// Mitsubishi GX Works2 project: china press #3 kontroller   PLC: Q04UDEH

// task MAIN (event TRUE, interval 0, priority 31): MAIN
// task MAIN1 (event TRUE, interval 0, priority 31): MAIN1_Block000
// task SFC (event TRUE, interval 0, priority 31): SFC_Block000, SFC_Block001, SFC_Block003, SFC_Block004, SFC_Block005, SFC_Block006

PROGRAM MAIN
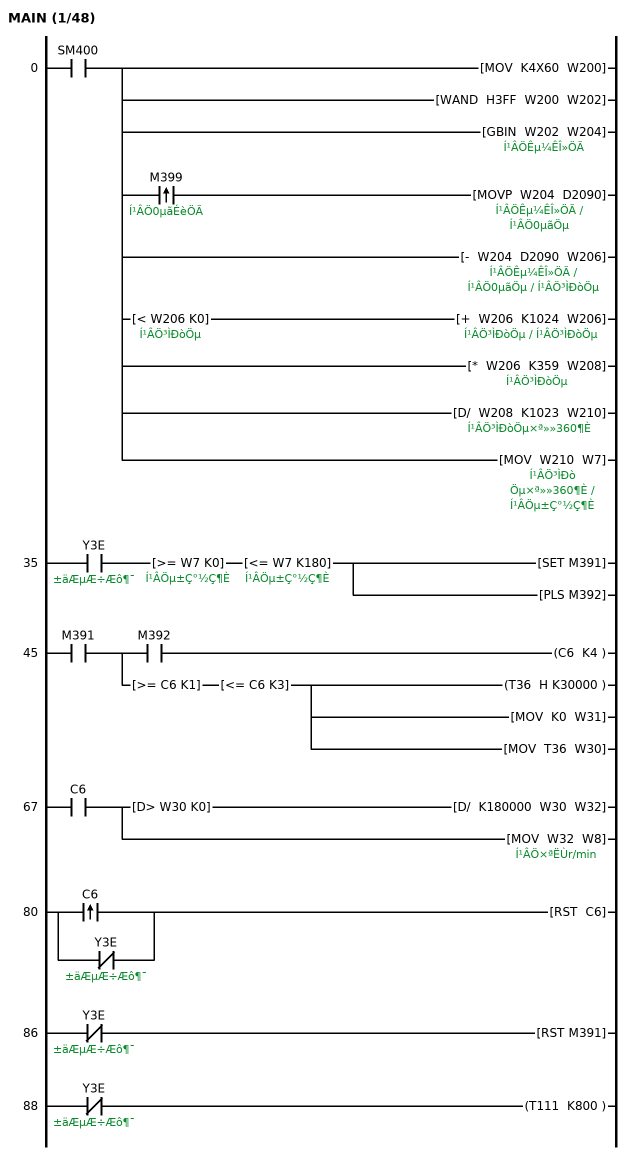
0     LD      SM400
      MOV     K4X60 W200  ; ¾øµØÖµ±àÂëÆ÷1
      WAND    H3FF W200 W202
      GBIN    W202 W204  ; Í¹ÂÖÊµ¼ÊÎ»ÖÃ
      MPS
      ANDP    M399  ; Í¹ÂÖ0µãÉèÖÃ
      MOVP    W204 D2090  ; Í¹ÂÖ0µãÖµ
      MPP
      -       W204 D2090 W206  ; Í¹ÂÖ³ÌÐòÖµ
      MPS
      AND<    W206 K0  ; Í¹ÂÖ³ÌÐòÖµ
      +       W206 K1024 W206
      MPP
      *       W206 K359 W208
      D/      W208 K1023 W210  ; Í¹ÂÖ³ÌÐòÖµ×ª»»360¶È
      MOV     W210 W7  ; Í¹ÂÖµ±Ç°½Ç¶È
35    LD      Y3E  ; ±äÆµÆ÷Æô¶¯
      AND>=   W7 K0  ; Í¹ÂÖµ±Ç°½Ç¶È
      AND<=   W7 K180  ; Í¹ÂÖµ±Ç°½Ç¶È
      SET     M391
      PLS     M392
45    LD      M391
      MPS
      AND     M392
      OUT     C6 K4
      MPP
      AND>=   C6 K1
      AND<=   C6 K3
      OUTH    T36 K30000
      MOV     K0 W31
      MOV     T36 W30
67    LD      C6
      MPS
      ANDD>   W30 K0
      D/      K180000 W30 W32
      MPP
      MOV     W32 W8  ; Í¹ÂÖ×ªËÙr/min
80    LDP     C6
      ORI     Y3E  ; ±äÆµÆ÷Æô¶¯
      RST     C6
86    LDI     Y3E  ; ±äÆµÆ÷Æô¶¯
      RST     M391
88    LDI     Y3E  ; ±äÆµÆ÷Æô¶¯
      OUT     T111 K800
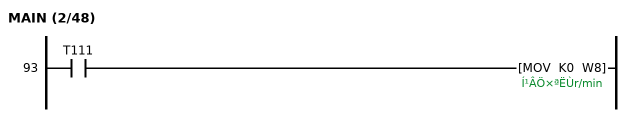
93    LD      T111
      MOV     K0 W8
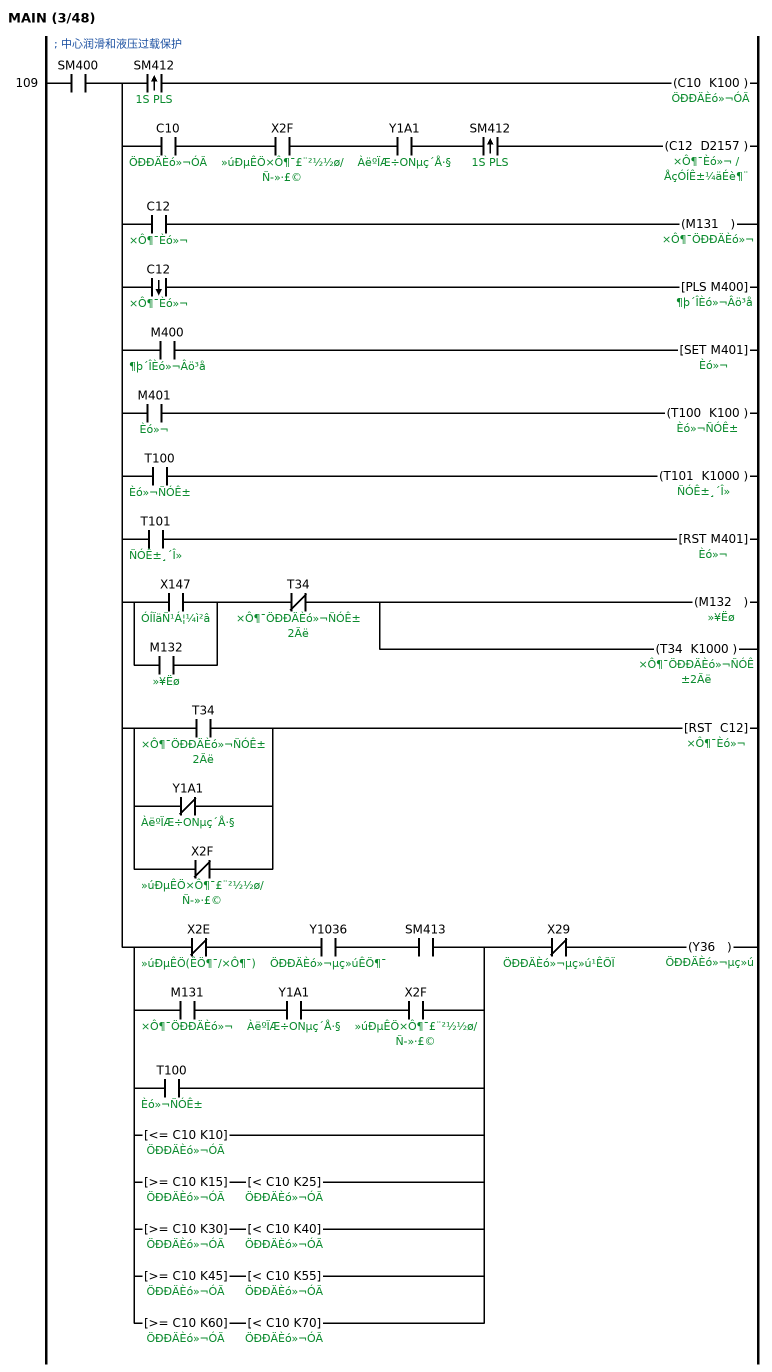
; 中心润滑和液压过载保护
109   LD      SM400
      MPS
      ANDP    SM412  ; 1S PLS
      OUT     C10 K100  ; ÖÐÐÄÈó»¬ÓÃ
      MRD
      AND     C10  ; ÖÐÐÄÈó»¬ÓÃ
      AND     X2F  ; »úÐµÊÖ×Ô¶¯£¨²½½ø/Ñ­»·£©
      AND     Y1A1  ; ÀëºÏÆ÷ONµç´Å·§
      ANDP    SM412  ; 1S PLS
      OUT     C12 D2157  ; ×Ô¶¯Èó»¬ / ÅçÓÍÊ±¼äÉè¶¨
      MRD
      AND     C12  ; ×Ô¶¯Èó»¬
      OUT     M131  ; ×Ô¶¯ÖÐÐÄÈó»¬
      MRD
      ANDF    C12  ; ×Ô¶¯Èó»¬
      PLS     M400  ; ¶þ´ÎÈó»¬Âö³å
      MRD
      AND     M400  ; ¶þ´ÎÈó»¬Âö³å
      SET     M401  ; Èó»¬
      MRD
      AND     M401  ; Èó»¬
      OUT     T100 K100  ; Èó»¬ÑÓÊ±
      MRD
      AND     T100  ; Èó»¬ÑÓÊ±
      OUT     T101 K1000  ; ÑÓÊ±¸´Î»
      MRD
      AND     T101  ; ÑÓÊ±¸´Î»
      RST     M401  ; Èó»¬
      MRD
      LD      X147  ; ÓÍÏäÑ¹Á¦¼ì²â
      OR      M132  ; »¥Ëø
      ANB
      ANI     T34  ; ×Ô¶¯ÖÐÐÄÈó»¬ÑÓÊ±2Ãë
      OUT     M132  ; »¥Ëø
      OUT     T34 K1000  ; ×Ô¶¯ÖÐÐÄÈó»¬ÑÓÊ±2Ãë
      MRD
      LD      T34  ; ×Ô¶¯ÖÐÐÄÈó»¬ÑÓÊ±2Ãë
      ORI     Y1A1  ; ÀëºÏÆ÷ONµç´Å·§
      ORI     X2F  ; »úÐµÊÖ×Ô¶¯£¨²½½ø/Ñ­»·£©
      ANB
      RST     C12  ; ×Ô¶¯Èó»¬
      MPP
      LDI     X2E  ; »úÐµÊÖ(ÊÖ¶¯/×Ô¶¯)
      AND     Y1036  ; ÖÐÐÄÈó»¬µç»úÊÖ¶¯
      AND     SM413
      LD      M131  ; ×Ô¶¯ÖÐÐÄÈó»¬
      AND     Y1A1  ; ÀëºÏÆ÷ONµç´Å·§
      AND     X2F  ; »úÐµÊÖ×Ô¶¯£¨²½½ø/Ñ­»·£©
      ORB
      OR      T100  ; Èó»¬ÑÓÊ±
      OR<=    C10 K10  ; ÖÐÐÄÈó»¬ÓÃ
      LD>=    C10 K15  ; ÖÐÐÄÈó»¬ÓÃ
      AND<    C10 K25  ; ÖÐÐÄÈó»¬ÓÃ
      ORB
      LD>=    C10 K30  ; ÖÐÐÄÈó»¬ÓÃ
      AND<    C10 K40  ; ÖÐÐÄÈó»¬ÓÃ
      ORB
      LD>=    C10 K45  ; ÖÐÐÄÈó»¬ÓÃ
      AND<    C10 K55  ; ÖÐÐÄÈó»¬ÓÃ
      ORB
      LD>=    C10 K60  ; ÖÐÐÄÈó»¬ÓÃ
      AND<    C10 K70  ; ÖÐÐÄÈó»¬ÓÃ
      ORB
      ANB
      ANI     X29  ; ÖÐÐÄÈó»¬µç»ú¹ÊÕÏ
      OUT     Y36  ; ÖÐÐÄÈó»¬µç»ú
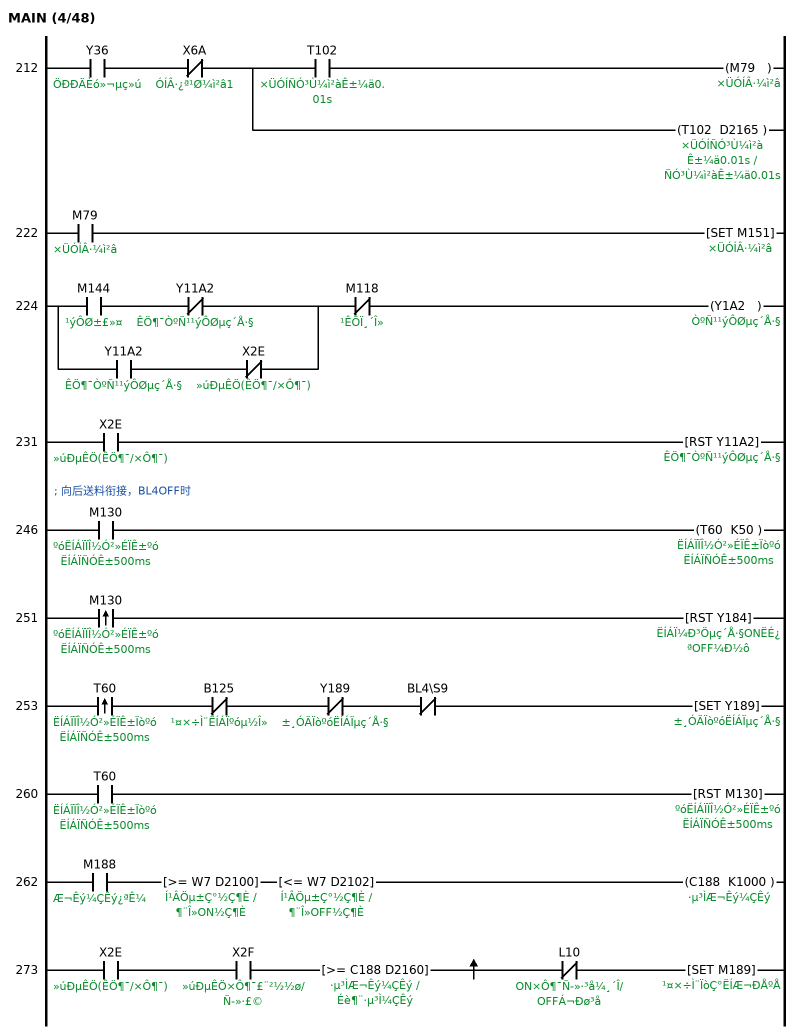
212   LD      Y36  ; ÖÐÐÄÈó»¬µç»ú
      ANI     X6A  ; ÓÍÂ·¿ª¹Ø¼ì²â1
      MPS
      AND     T102  ; ×ÜÓÍÑÓ³Ù¼ì²àÊ±¼ä0.01s
      OUT     M79  ; ×ÜÓÍÂ·¼ì²â
      MPP
      OUT     T102 D2165  ; ×ÜÓÍÑÓ³Ù¼ì²àÊ±¼ä0.01s / ÑÓ³Ù¼ì²àÊ±¼ä0.01s
222   LD      M79  ; ×ÜÓÍÂ·¼ì²â
      SET     M151  ; ×ÜÓÍÂ·¼ì²â
224   LD      M144  ; ¹ýÔØ±£»¤
      ANI     Y11A2  ; ÊÖ¶¯ÒºÑ¹¹ýÔØµç´Å·§
      LD      Y11A2  ; ÊÖ¶¯ÒºÑ¹¹ýÔØµç´Å·§
      ANI     X2E  ; »úÐµÊÖ(ÊÖ¶¯/×Ô¶¯)
      ORB
      ANI     M118  ; ¹ÊÕÏ¸´Î»
      OUT     Y1A2  ; ÒºÑ¹¹ýÔØµç´Å·§
231   LD      X2E  ; »úÐµÊÖ(ÊÖ¶¯/×Ô¶¯)
      RST     Y11A2  ; ÊÖ¶¯ÒºÑ¹¹ýÔØµç´Å·§
; 向后送料衔接，BL4OFF时
246   LD      M130  ; ºóËÍÁÏÏÎ½Ó²»ÉÏÊ±ºóËÍÁÏÑÓÊ±500ms
      OUT     T60 K50  ; ËÍÁÏÏÎ½Ó²»ÉÏÊ±ÏòºóËÍÁÏÑÓÊ±500ms
251   LDP     M130  ; ºóËÍÁÏÏÎ½Ó²»ÉÏÊ±ºóËÍÁÏÑÓÊ±500ms
      RST     Y184  ; ËÍÁÏ¼Ð³Öµç´Å·§ONËÉ¿ªOFF¼Ð½ô
253   LDP     T60  ; ËÍÁÏÏÎ½Ó²»ÉÏÊ±ÏòºóËÍÁÏÑÓÊ±500ms
      ANI     B125  ; ¹¤×÷Ì¨ËÍÁÏºóµ½Î»
      ANI     Y189  ; ±¸ÓÃÏòºóËÍÁÏµç´Å·§
      ANI     BL4\S9
      SET     Y189  ; ±¸ÓÃÏòºóËÍÁÏµç´Å·§
260   LD      T60  ; ËÍÁÏÏÎ½Ó²»ÉÏÊ±ÏòºóËÍÁÏÑÓÊ±500ms
      RST     M130  ; ºóËÍÁÏÏÎ½Ó²»ÉÏÊ±ºóËÍÁÏÑÓÊ±500ms
262   LD      M188  ; Æ¬Êý¼ÇÊý¿ªÊ¼
      AND>=   W7 D2100  ; Í¹ÂÖµ±Ç°½Ç¶È / ¶¨Î»ON½Ç¶È
      AND<=   W7 D2102  ; Í¹ÂÖµ±Ç°½Ç¶È / ¶¨Î»OFF½Ç¶È
      OUT     C188 K1000  ; ·µ³ÌÆ¬Êý¼ÇÊý
273   LD      X2E  ; »úÐµÊÖ(ÊÖ¶¯/×Ô¶¯)
      AND     X2F  ; »úÐµÊÖ×Ô¶¯£¨²½½ø/Ñ­»·£©
      AND>=   C188 D2160  ; ·µ³ÌÆ¬Êý¼ÇÊý / Éè¶¨·µ³Ì¼ÇÊý
      MEP
      ANI     L10  ; ON×Ô¶¯Ñ­»·³å¼¸´Î/OFFÁ¬Ðø³å
      SET     M189  ; ¹¤×÷Ì¨ÏòÇ°ËÍÆ¬ÐÅºÅ
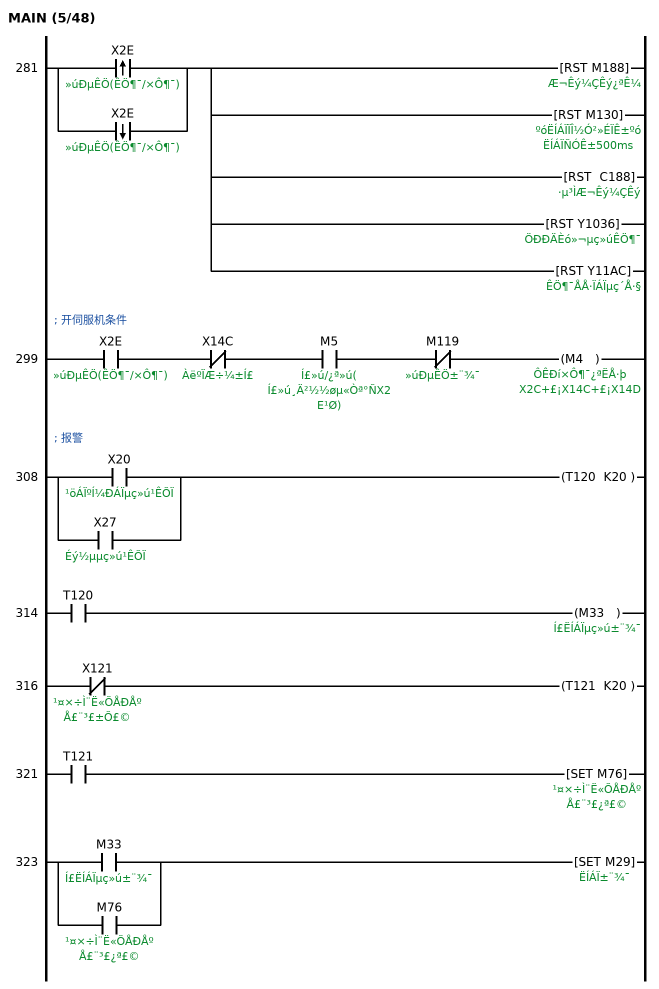
281   LDP     X2E  ; »úÐµÊÖ(ÊÖ¶¯/×Ô¶¯)
      ORF     X2E  ; »úÐµÊÖ(ÊÖ¶¯/×Ô¶¯)
      RST     M188  ; Æ¬Êý¼ÇÊý¿ªÊ¼
      RST     M130  ; ºóËÍÁÏÏÎ½Ó²»ÉÏÊ±ºóËÍÁÏÑÓÊ±500ms
      RST     C188  ; ·µ³ÌÆ¬Êý¼ÇÊý
      RST     Y1036  ; ÖÐÐÄÈó»¬µç»úÊÖ¶¯
      RST     Y11AC  ; ÊÖ¶¯ÅÅ·ÏÁÏµç´Å·§
; 开伺服机条件
299   LD      X2E  ; »úÐµÊÖ(ÊÖ¶¯/×Ô¶¯)
      ANI     X14C  ; ÀëºÏÆ÷¼±Í£
      AND     M5  ; Í£»ú/¿ª»ú(Í£»ú¸Ä²½½øµ«Òª°ÑX2E¹Ø)
      ANI     M119  ; »úÐµÊÖ±¨¾¯
      OUT     M4  ; ÔÊÐí×Ô¶¯¿ªËÅ·þX2C+£¡X14C+£¡X14D
; 报警
308   LD      X20  ; ¹öÁÏºÍ¼ÐÁÏµç»ú¹ÊÕÏ
      OR      X27  ; Éý½µµç»ú¹ÊÕÏ
      OUT     T120 K20
314   LD      T120
      OUT     M33  ; Í£ËÍÁÏµç»ú±¨¾¯
316   LDI     X121  ; ¹¤×÷Ì¨Ë«ÕÅÐÅºÅ£¨³£±Õ£©
      OUT     T121 K20
321   LD      T121
      SET     M76  ; ¹¤×÷Ì¨Ë«ÕÅÐÅºÅ£¨³£¿ª£©
323   LD      M33  ; Í£ËÍÁÏµç»ú±¨¾¯
      OR      M76  ; ¹¤×÷Ì¨Ë«ÕÅÐÅºÅ£¨³£¿ª£©
      SET     M29  ; ËÍÁÏ±¨¾¯
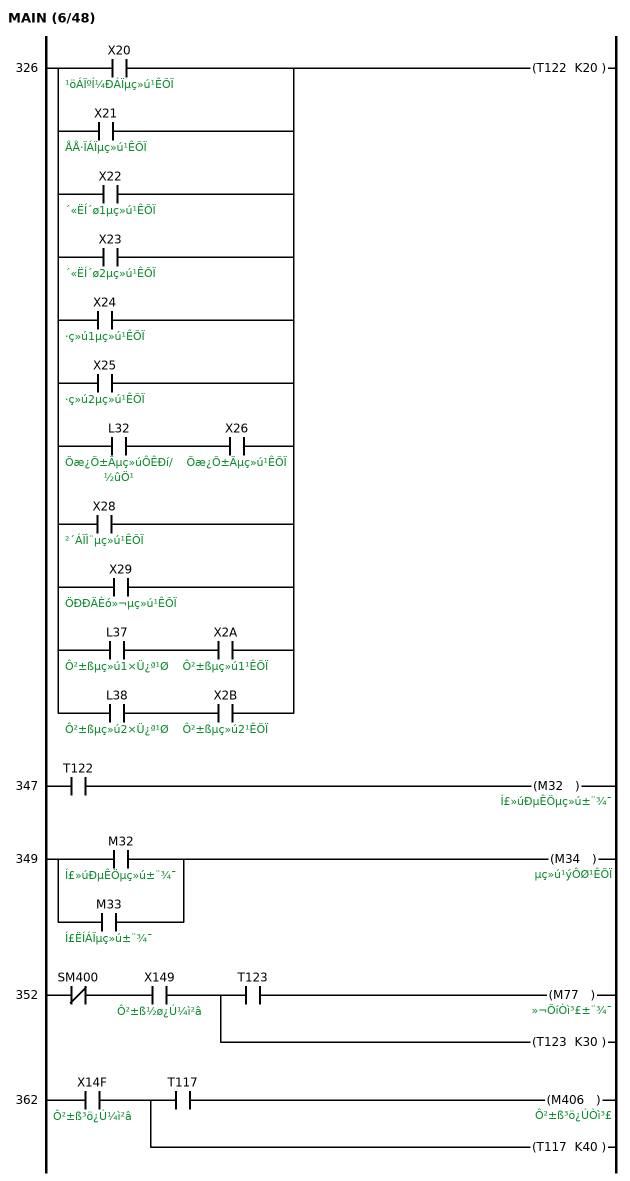
326   LD      X20  ; ¹öÁÏºÍ¼ÐÁÏµç»ú¹ÊÕÏ
      OR      X21  ; ÅÅ·ÏÁÏµç»ú¹ÊÕÏ
      OR      X22  ; ´«ËÍ´ø1µç»ú¹ÊÕÏ
      OR      X23  ; ´«ËÍ´ø2µç»ú¹ÊÕÏ
      OR      X24  ; ·ç»ú1µç»ú¹ÊÕÏ
      OR      X25  ; ·ç»ú2µç»ú¹ÊÕÏ
      LD      L32  ; Õæ¿Õ±Ãµç»úÔÊÐí/½ûÖ¹
      AND     X26  ; Õæ¿Õ±Ãµç»ú¹ÊÕÏ
      ORB
      OR      X28  ; ²´ÁÏÌ¨µç»ú¹ÊÕÏ
      OR      X29  ; ÖÐÐÄÈó»¬µç»ú¹ÊÕÏ
      LD      L37  ; Ô²±ßµç»ú1×Ü¿ª¹Ø
      AND     X2A  ; Ô²±ßµç»ú1¹ÊÕÏ
      ORB
      LD      L38  ; Ô²±ßµç»ú2×Ü¿ª¹Ø
      AND     X2B  ; Ô²±ßµç»ú2¹ÊÕÏ
      ORB
      OUT     T122 K20
347   LD      T122
      OUT     M32  ; Í£»úÐµÊÖµç»ú±¨¾¯
349   LD      M32  ; Í£»úÐµÊÖµç»ú±¨¾¯
      OR      M33  ; Í£ËÍÁÏµç»ú±¨¾¯
      OUT     M34  ; µç»ú¹ýÔØ¹ÊÕÏ
352   LDI     SM400
      AND     X149  ; Ô²±ß½ø¿Ú¼ì²â
      MPS
      AND     T123
      OUT     M77  ; »¬ÕíÒì³£±¨¾¯
      MPP
      OUT     T123 K30
362   LD      X14F  ; Ô²±ß³ö¿Ú¼ì²â
      MPS
      AND     T117
      OUT     M406  ; Ô²±ß³ö¿ÚÒì³£
      MPP
      OUT     T117 K40
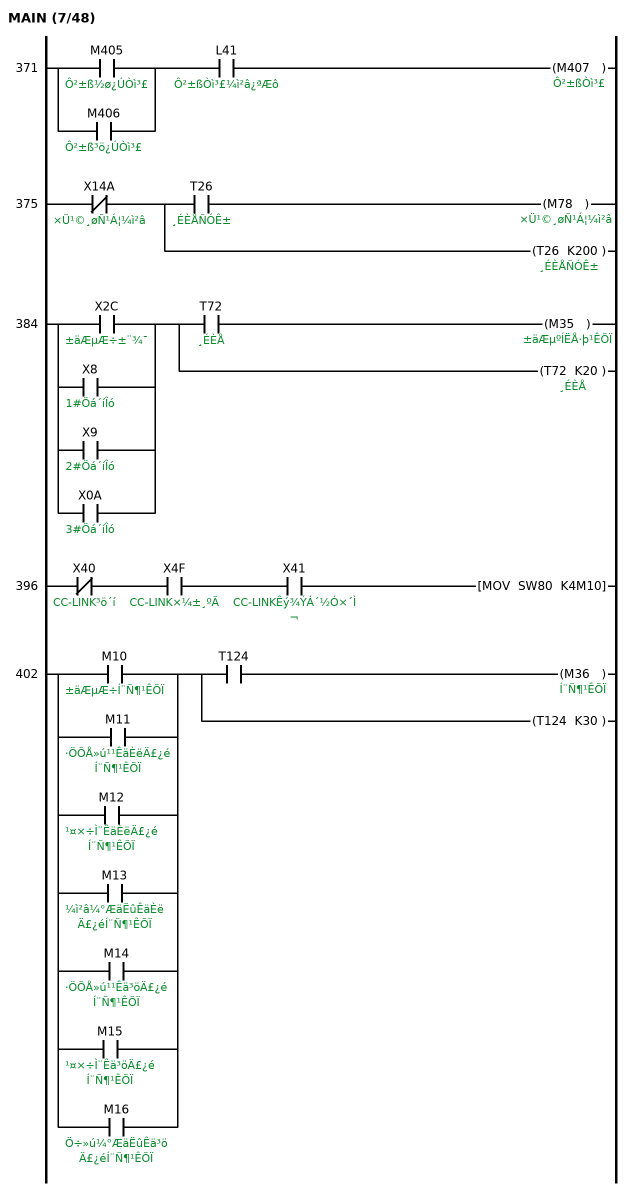
371   LD      M405  ; Ô²±ß½ø¿ÚÒì³£
      OR      M406  ; Ô²±ß³ö¿ÚÒì³£
      AND     L41  ; Ô²±ßÒì³£¼ì²â¿ªÆô
      OUT     M407  ; Ô²±ßÒì³£
375   LDI     X14A  ; ×Ü¹©¸øÑ¹Á¦¼ì²â
      MPS
      AND     T26  ; ¸ÉÈÅÑÓÊ±
      OUT     M78  ; ×Ü¹©¸øÑ¹Á¦¼ì²â
      MPP
      OUT     T26 K200  ; ¸ÉÈÅÑÓÊ±
384   LD      X2C  ; ±äÆµÆ÷±¨¾¯
      OR      X8  ; 1#Öá´íÎó
      OR      X9  ; 2#Öá´íÎó
      OR      X0A  ; 3#Öá´íÎó
      MPS
      AND     T72  ; ¸ÉÈÅ
      OUT     M35  ; ±äÆµºÍËÅ·þ¹ÊÕÏ
      MPP
      OUT     T72 K20  ; ¸ÉÈÅ
396   LDI     X40  ; CC-LINK³ö´í
      AND     X4F  ; CC-LINK×¼±¸ºÃ
      AND     X41  ; CC-LINKÊý¾ÝÁ´½Ó×´Ì¬
      MOV     SW80 K4M10  ; ±äÆµÆ÷Í¨Ñ¶¹ÊÕÏ
402   LD      M10  ; ±äÆµÆ÷Í¨Ñ¶¹ÊÕÏ
      OR      M11  ; ·ÖÕÅ»ú¹¹ÊäÈëÄ£¿éÍ¨Ñ¶¹ÊÕÏ
      OR      M12  ; ¹¤×÷Ì¨ÊäÈëÄ£¿éÍ¨Ñ¶¹ÊÕÏ
      OR      M13  ; ¼ì²â¼°ÆäËûÊäÈëÄ£¿éÍ¨Ñ¶¹ÊÕÏ
      OR      M14  ; ·ÖÕÅ»ú¹¹Êä³öÄ£¿éÍ¨Ñ¶¹ÊÕÏ
      OR      M15  ; ¹¤×÷Ì¨Êä³öÄ£¿éÍ¨Ñ¶¹ÊÕÏ
      OR      M16  ; Ö÷»ú¼°ÆäËûÊä³öÄ£¿éÍ¨Ñ¶¹ÊÕÏ
      MPS
      AND     T124
      OUT     M36  ; Í¨Ñ¶¹ÊÕÏ
      MPP
      OUT     T124 K30
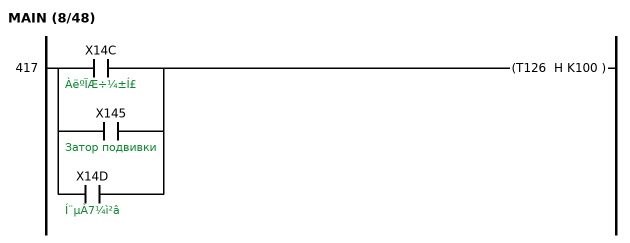
417   LD      X14C  ; ÀëºÏÆ÷¼±Í£
      OR      X145  ; Затор подвивки
      OR      X14D  ; Í¨µÀ7¼ì²â
      OUTH    T126 K100
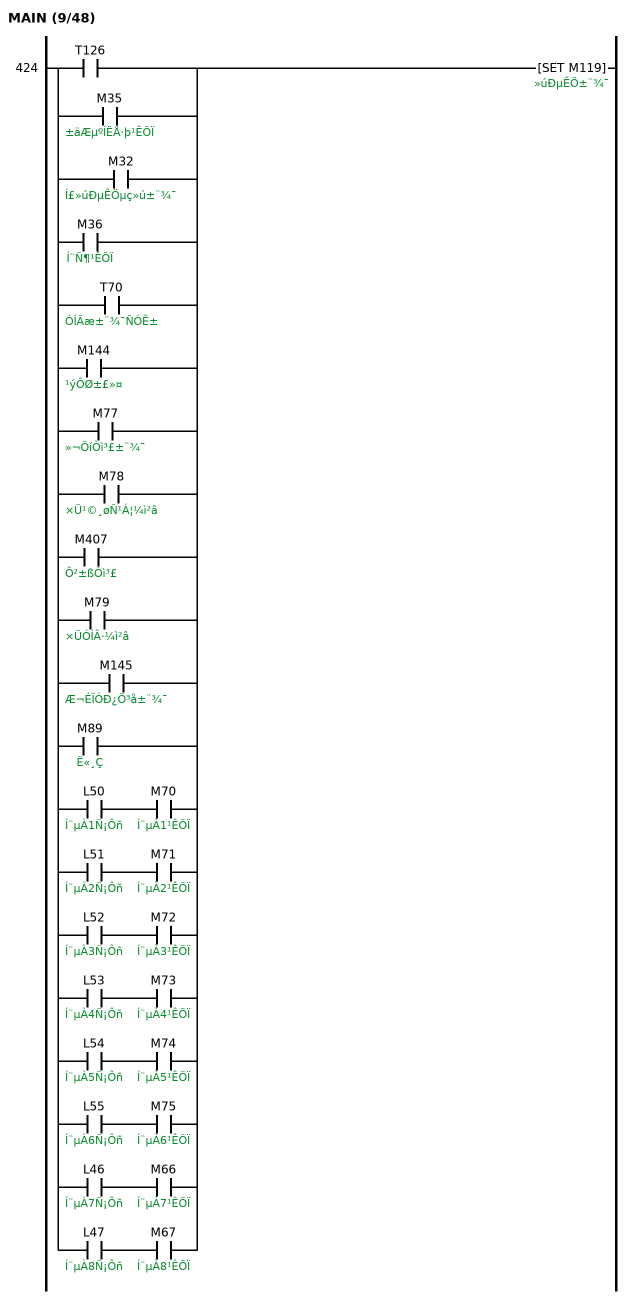
424   LD      T126
      OR      M35  ; ±äÆµºÍËÅ·þ¹ÊÕÏ
      OR      M32  ; Í£»úÐµÊÖµç»ú±¨¾¯
      OR      M36  ; Í¨Ñ¶¹ÊÕÏ
      OR      T70  ; ÓÍÃæ±¨¾¯ÑÓÊ±
      OR      M144  ; ¹ýÔØ±£»¤
      OR      M77  ; »¬ÕíÒì³£±¨¾¯
      OR      M78  ; ×Ü¹©¸øÑ¹Á¦¼ì²â
      OR      M407  ; Ô²±ßÒì³£
      OR      M79  ; ×ÜÓÍÂ·¼ì²â
      OR      M145  ; Æ¬ÉÏÓÐ¿Õ³å±¨¾¯
      OR      M89  ; Ë«¸Ç
      LD      L50  ; Í¨µÀ1Ñ¡Ôñ
      AND     M70  ; Í¨µÀ1¹ÊÕÏ
      ORB
      LD      L51  ; Í¨µÀ2Ñ¡Ôñ
      AND     M71  ; Í¨µÀ2¹ÊÕÏ
      ORB
      LD      L52  ; Í¨µÀ3Ñ¡Ôñ
      AND     M72  ; Í¨µÀ3¹ÊÕÏ
      ORB
      LD      L53  ; Í¨µÀ4Ñ¡Ôñ
      AND     M73  ; Í¨µÀ4¹ÊÕÏ
      ORB
      LD      L54  ; Í¨µÀ5Ñ¡Ôñ
      AND     M74  ; Í¨µÀ5¹ÊÕÏ
      ORB
      LD      L55  ; Í¨µÀ6Ñ¡Ôñ
      AND     M75  ; Í¨µÀ6¹ÊÕÏ
      ORB
      LD      L46  ; Í¨µÀ7Ñ¡Ôñ
      AND     M66  ; Í¨µÀ7¹ÊÕÏ
      ORB
      LD      L47  ; Í¨µÀ8Ñ¡Ôñ
      AND     M67  ; Í¨µÀ8¹ÊÕÏ
      ORB
      SET     M119  ; »úÐµÊÖ±¨¾¯
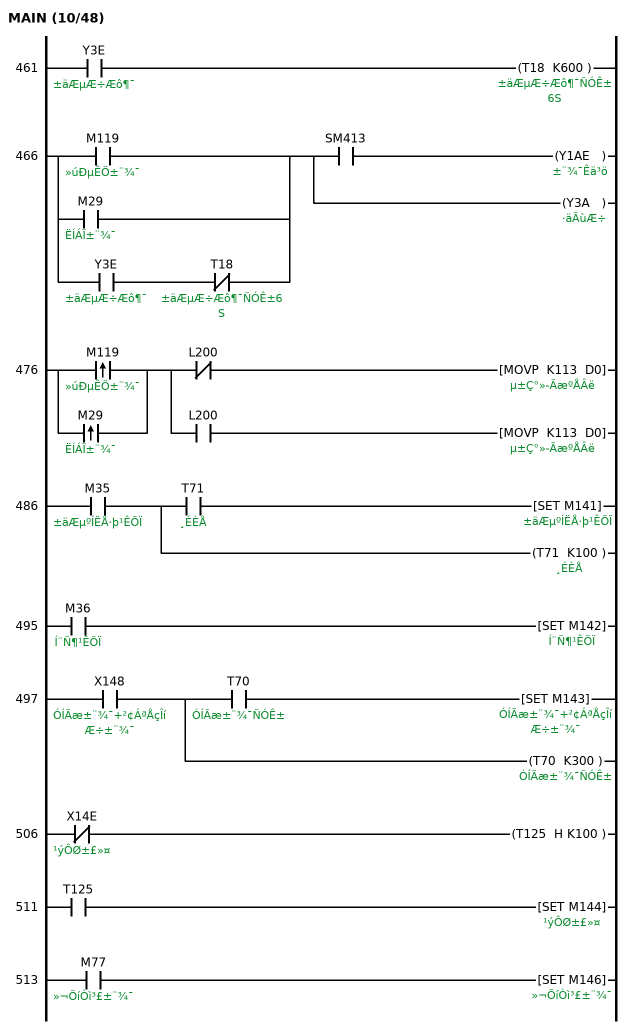
461   LD      Y3E  ; ±äÆµÆ÷Æô¶¯
      OUT     T18 K600  ; ±äÆµÆ÷Æô¶¯ÑÓÊ±6S
466   LD      M119  ; »úÐµÊÖ±¨¾¯
      OR      M29  ; ËÍÁÏ±¨¾¯
      LD      Y3E  ; ±äÆµÆ÷Æô¶¯
      ANI     T18  ; ±äÆµÆ÷Æô¶¯ÑÓÊ±6S
      ORB
      MPS
      AND     SM413
      OUT     Y1AE  ; ±¨¾¯Êä³ö
      MPP
      OUT     Y3A  ; ·äÃùÆ÷
476   LDP     M119  ; »úÐµÊÖ±¨¾¯
      ORP     M29  ; ËÍÁÏ±¨¾¯
      MPS
      ANI     L200
      MOVP    K113 D0  ; µ±Ç°»­ÃæºÅÂë
      MPP
      AND     L200
      MOVP    K113 D0
486   LD      M35  ; ±äÆµºÍËÅ·þ¹ÊÕÏ
      MPS
      AND     T71  ; ¸ÉÈÅ
      SET     M141  ; ±äÆµºÍËÅ·þ¹ÊÕÏ
      MPP
      OUT     T71 K100  ; ¸ÉÈÅ
495   LD      M36  ; Í¨Ñ¶¹ÊÕÏ
      SET     M142  ; Í¨Ñ¶¹ÊÕÏ
497   LD      X148  ; ÓÍÃæ±¨¾¯+²¢ÁªÅçÎíÆ÷±¨¾¯
      MPS
      AND     T70  ; ÓÍÃæ±¨¾¯ÑÓÊ±
      SET     M143  ; ÓÍÃæ±¨¾¯+²¢ÁªÅçÎíÆ÷±¨¾¯
      MPP
      OUT     T70 K300  ; ÓÍÃæ±¨¾¯ÑÓÊ±
506   LDI     X14E  ; ¹ýÔØ±£»¤
      OUTH    T125 K100
511   LD      T125
      SET     M144  ; ¹ýÔØ±£»¤
513   LD      M77  ; »¬ÕíÒì³£±¨¾¯
      SET     M146  ; »¬ÕíÒì³£±¨¾¯
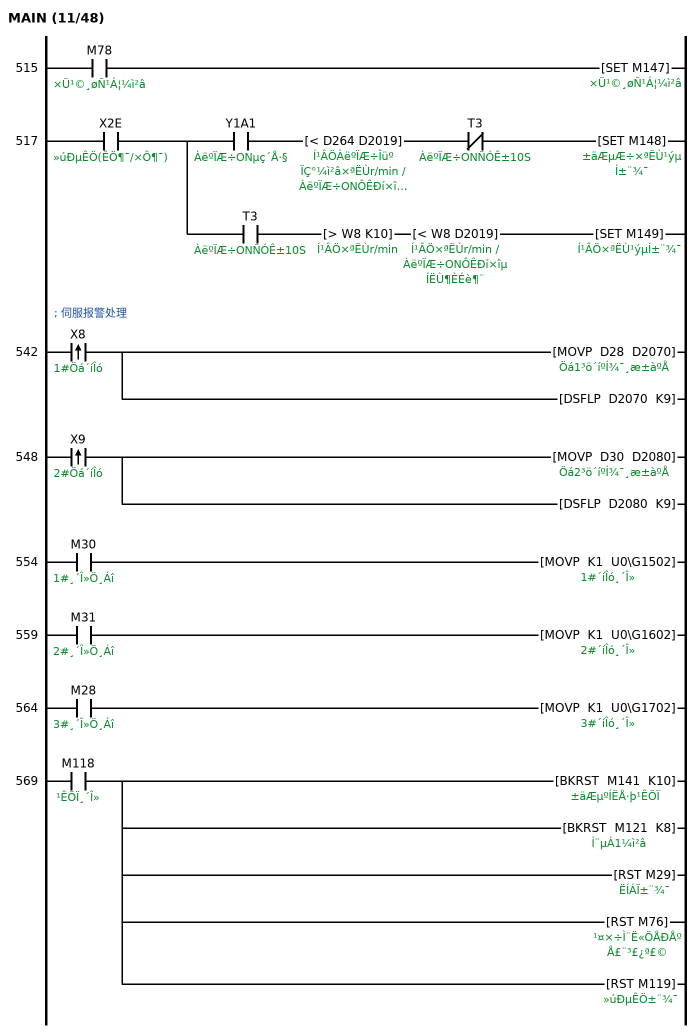
515   LD      M78  ; ×Ü¹©¸øÑ¹Á¦¼ì²â
      SET     M147  ; ×Ü¹©¸øÑ¹Á¦¼ì²â
517   LD      X2E  ; »úÐµÊÖ(ÊÖ¶¯/×Ô¶¯)
      MPS
      AND     Y1A1  ; ÀëºÏÆ÷ONµç´Å·§
      AND<    D264 D2019  ; Í¹ÂÖÀëºÏÆ÷ÎüºÏÇ°¼ì²â×ªËÙr/min / ÀëºÏÆ÷ONÔÊÐí×îµÍËÙ¶ÈÉè¶¨
      ANI     T3  ; ÀëºÏÆ÷ONÑÓÊ±10S
      SET     M148  ; ±äÆµÆ÷×ªËÙ¹ýµÍ±¨¾¯
      MPP
      AND     T3  ; ÀëºÏÆ÷ONÑÓÊ±10S
      AND>    W8 K10  ; Í¹ÂÖ×ªËÙr/min
      AND<    W8 D2019  ; Í¹ÂÖ×ªËÙr/min / ÀëºÏÆ÷ONÔÊÐí×îµÍËÙ¶ÈÉè¶¨
      SET     M149  ; Í¹ÂÖ×ªËÙ¹ýµÍ±¨¾¯
; 伺服报警处理
542   LDP     X8  ; 1#Öá´íÎó
      MOVP    D28 D2070  ; Öá1³ö´íºÍ¾¯¸æ±àºÅ
      DSFLP   D2070 K9
548   LDP     X9  ; 2#Öá´íÎó
      MOVP    D30 D2080  ; Öá2³ö´íºÍ¾¯¸æ±àºÅ
      DSFLP   D2080 K9
554   LD      M30  ; 1#¸´Î»Ö¸Áî
      MOVP    K1 U0\G1502  ; 1#´íÎó¸´Î»
559   LD      M31  ; 2#¸´Î»Ö¸Áî
      MOVP    K1 U0\G1602  ; 2#´íÎó¸´Î»
564   LD      M28  ; 3#¸´Î»Ö¸Áî
      MOVP    K1 U0\G1702  ; 3#´íÎó¸´Î»
569   LD      M118  ; ¹ÊÕÏ¸´Î»
      BKRST   M141 K10
      BKRST   M121 K8  ; Í¨µÀ1¼ì²â
      RST     M29  ; ËÍÁÏ±¨¾¯
      RST     M76  ; ¹¤×÷Ì¨Ë«ÕÅÐÅºÅ£¨³£¿ª£©
      RST     M119  ; »úÐµÊÖ±¨¾¯
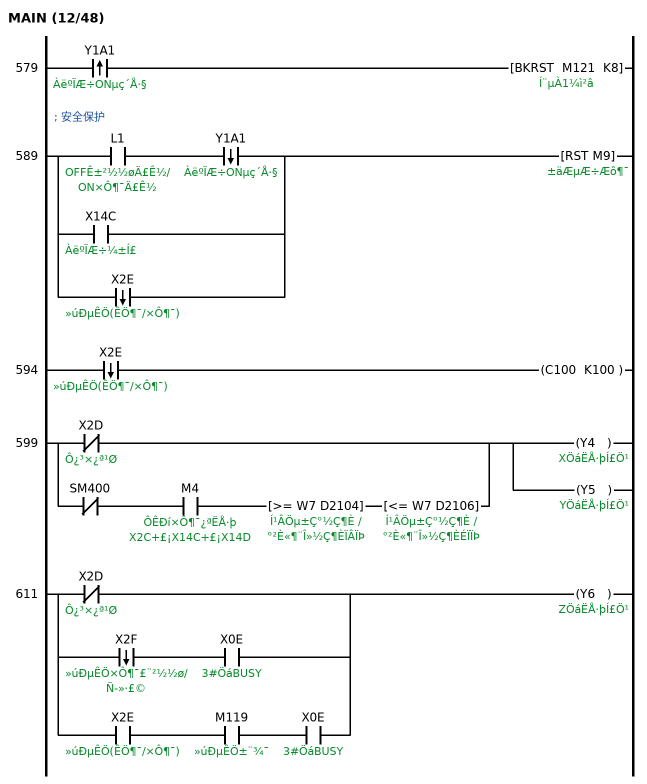
579   LDP     Y1A1  ; ÀëºÏÆ÷ONµç´Å·§
      BKRST   M121 K8
; 安全保护
589   LD      L1  ; OFFÊ±²½½øÄ£Ê½/ON×Ô¶¯Ä£Ê½
      ANDF    Y1A1  ; ÀëºÏÆ÷ONµç´Å·§
      OR      X14C  ; ÀëºÏÆ÷¼±Í£
      ORF     X2E  ; »úÐµÊÖ(ÊÖ¶¯/×Ô¶¯)
      RST     M9  ; ±äÆµÆ÷Æô¶¯
594   LDF     X2E  ; »úÐµÊÖ(ÊÖ¶¯/×Ô¶¯)
      OUT     C100 K100
599   LDI     X2D  ; Ô¿³×¿ª¹Ø
      LDI     SM400
      AND     M4  ; ÔÊÐí×Ô¶¯¿ªËÅ·þX2C+£¡X14C+£¡X14D
      AND>=   W7 D2104  ; Í¹ÂÖµ±Ç°½Ç¶È / °²È«¶¨Î»½Ç¶ÈÏÂÏÞ
      AND<=   W7 D2106  ; Í¹ÂÖµ±Ç°½Ç¶È / °²È«¶¨Î»½Ç¶ÈÉÏÏÞ
      ORB
      OUT     Y4  ; XÖáËÅ·þÍ£Ö¹
      OUT     Y5  ; YÖáËÅ·þÍ£Ö¹
611   LDI     X2D  ; Ô¿³×¿ª¹Ø
      LDF     X2F  ; »úÐµÊÖ×Ô¶¯£¨²½½ø/Ñ­»·£©
      AND     X0E  ; 3#ÖáBUSY
      ORB
      LD      X2E  ; »úÐµÊÖ(ÊÖ¶¯/×Ô¶¯)
      AND     M119  ; »úÐµÊÖ±¨¾¯
      AND     X0E  ; 3#ÖáBUSY
      ORB
      OUT     Y6  ; ZÖáËÅ·þÍ£Ö¹
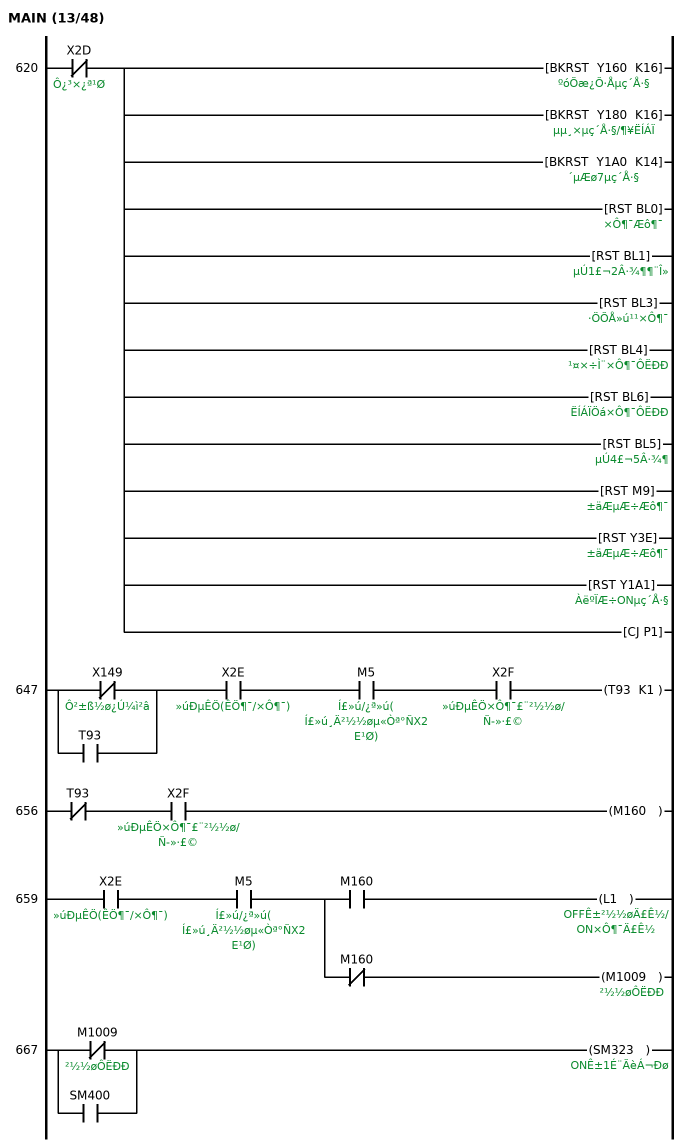
620   LDI     X2D  ; Ô¿³×¿ª¹Ø
      BKRST   Y160 K16  ; ºóÕæ¿Õ·Åµç´Å·§
      BKRST   Y180 K16  ; µµ¸×µç´Å·§/¶¥ËÍÁÏ
      BKRST   Y1A0 K14  ; ´µÆø7µç´Å·§
      RST     BL0  ; ×Ô¶¯Æô¶¯
      RST     BL1  ; µÚ1£¬2Â·¾¶¶¨Î»
      RST     BL3  ; ·ÖÕÅ»ú¹¹×Ô¶¯
      RST     BL4  ; ¹¤×÷Ì¨×Ô¶¯ÔËÐÐ
      RST     BL6  ; ËÍÁÏÖá×Ô¶¯ÔËÐÐ
      RST     BL5  ; µÚ4£¬5Â·¾¶
      RST     M9  ; ±äÆµÆ÷Æô¶¯
      RST     Y3E  ; ±äÆµÆ÷Æô¶¯
      RST     Y1A1  ; ÀëºÏÆ÷ONµç´Å·§
      CJ      P1
647   LDI     X149  ; Ô²±ß½ø¿Ú¼ì²â
      OR      T93
      AND     X2E  ; »úÐµÊÖ(ÊÖ¶¯/×Ô¶¯)
      AND     M5  ; Í£»ú/¿ª»ú(Í£»ú¸Ä²½½øµ«Òª°ÑX2E¹Ø)
      AND     X2F  ; »úÐµÊÖ×Ô¶¯£¨²½½ø/Ñ­»·£©
      OUT     T93 K1
656   LDI     T93
      AND     X2F  ; »úÐµÊÖ×Ô¶¯£¨²½½ø/Ñ­»·£©
      OUT     M160
659   LD      X2E  ; »úÐµÊÖ(ÊÖ¶¯/×Ô¶¯)
      AND     M5  ; Í£»ú/¿ª»ú(Í£»ú¸Ä²½½øµ«Òª°ÑX2E¹Ø)
      MPS
      AND     M160
      OUT     L1  ; OFFÊ±²½½øÄ£Ê½/ON×Ô¶¯Ä£Ê½
      MPP
      ANI     M160
      OUT     M1009  ; ²½½øÔËÐÐ
667   LDI     M1009  ; ²½½øÔËÐÐ
      OR      SM400
      OUT     SM323  ; ONÊ±1É¨ÃèÁ¬Ðø
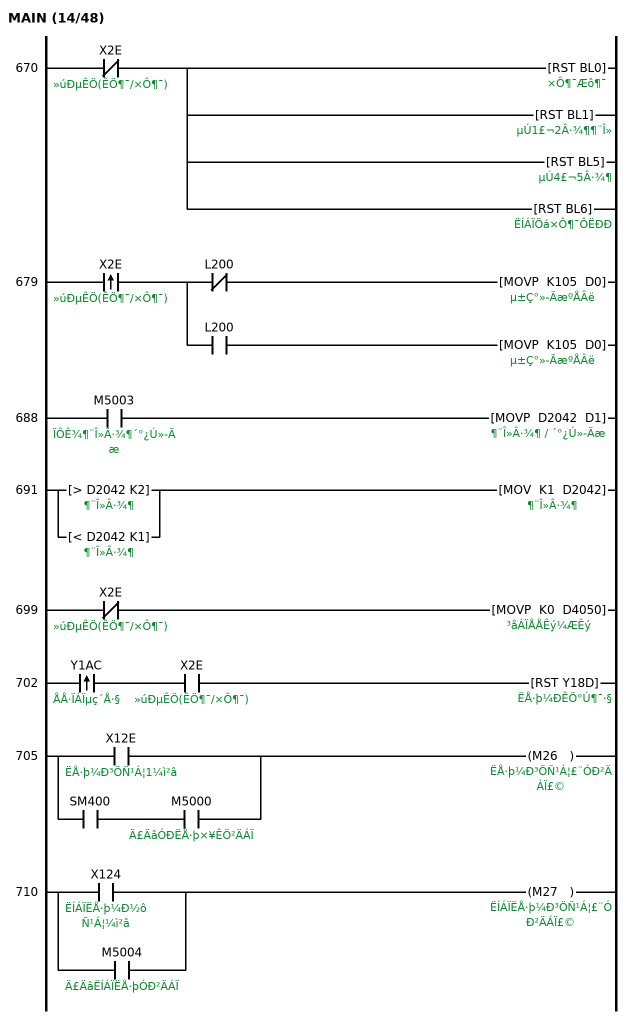
670   LDI     X2E  ; »úÐµÊÖ(ÊÖ¶¯/×Ô¶¯)
      RST     BL0  ; ×Ô¶¯Æô¶¯
      RST     BL1  ; µÚ1£¬2Â·¾¶¶¨Î»
      RST     BL5  ; µÚ4£¬5Â·¾¶
      RST     BL6  ; ËÍÁÏÖá×Ô¶¯ÔËÐÐ
679   LDP     X2E  ; »úÐµÊÖ(ÊÖ¶¯/×Ô¶¯)
      MPS
      ANI     L200
      MOVP    K105 D0
      MPP
      AND     L200
      MOVP    K105 D0
688   LD      M5003  ; ÏÔÊ¾¶¨Î»Â·¾¶´°¿Ú»­Ãæ
      MOVP    D2042 D1  ; ¶¨Î»Â·¾¶ / ´°¿Ú»­Ãæ
691   LD>     D2042 K2  ; ¶¨Î»Â·¾¶
      OR<     D2042 K1  ; ¶¨Î»Â·¾¶
      MOV     K1 D2042
699   LDI     X2E  ; »úÐµÊÖ(ÊÖ¶¯/×Ô¶¯)
      MOVP    K0 D4050  ; ³åÁÏÅÅÊý¼ÆÊý
702   LDP     Y1AC  ; ÅÅ·ÏÁÏµç´Å·§
      AND     X2E  ; »úÐµÊÖ(ÊÖ¶¯/×Ô¶¯)
      RST     Y18D  ; ËÅ·þ¼ÐÊÖ°Ú¶¯·§
705   LD      X12E  ; ËÅ·þ¼Ð³ÖÑ¹Á¦1¼ì²â
      LD      SM400
      AND     M5000  ; Ä£ÄâÓÐËÅ·þ×¥ÊÖ²ÄÁÏ
      ORB
      OUT     M26  ; ËÅ·þ¼Ð³ÖÑ¹Á¦£¨ÓÐ²ÄÁÏ£©
710   LD      X124  ; ËÍÁÏËÅ·þ¼Ð½ôÑ¹Á¦¼ì²â
      OR      M5004  ; Ä£ÄâËÍÁÏËÅ·þÓÐ²ÄÁÏ
      OUT     M27  ; ËÍÁÏËÅ·þ¼Ð³ÖÑ¹Á¦£¨ÓÐ²ÄÁÏ£©
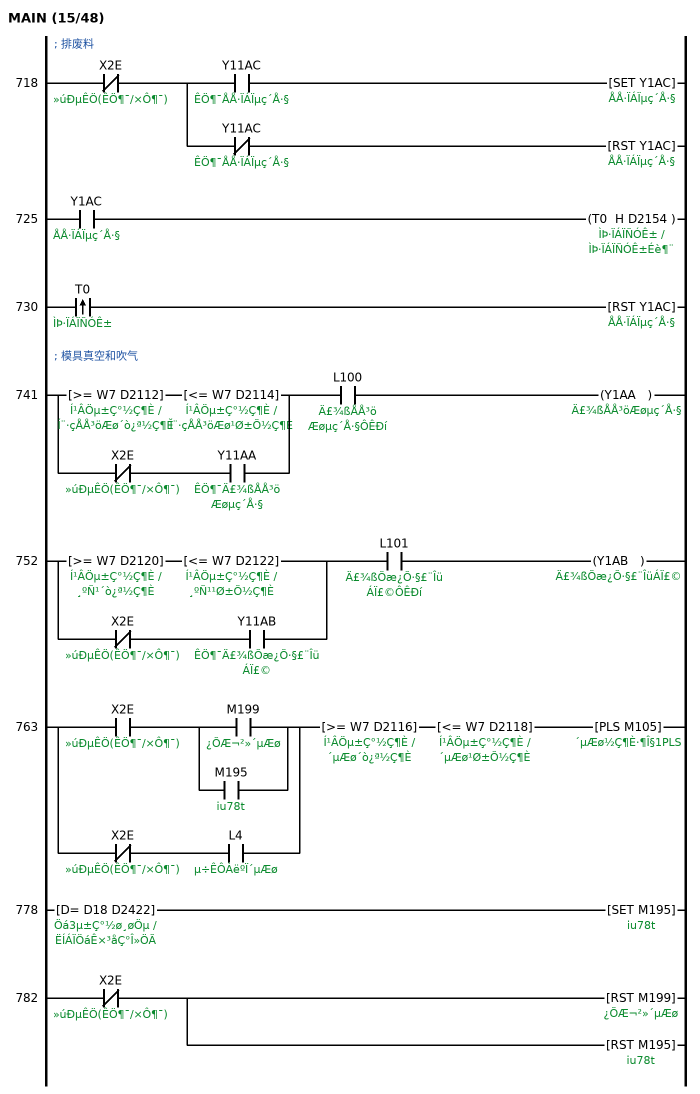
; 排废料
718   LDI     X2E  ; »úÐµÊÖ(ÊÖ¶¯/×Ô¶¯)
      MPS
      AND     Y11AC  ; ÊÖ¶¯ÅÅ·ÏÁÏµç´Å·§
      SET     Y1AC  ; ÅÅ·ÏÁÏµç´Å·§
      MPP
      ANI     Y11AC  ; ÊÖ¶¯ÅÅ·ÏÁÏµç´Å·§
      RST     Y1AC  ; ÅÅ·ÏÁÏµç´Å·§
725   LD      Y1AC  ; ÅÅ·ÏÁÏµç´Å·§
      OUTH    T0 D2154  ; ÌÞ·ÏÁÏÑÓÊ± / ÌÞ·ÏÁÏÑÓÊ±Éè¶¨
730   LDP     T0  ; ÌÞ·ÏÁÏÑÓÊ±
      RST     Y1AC  ; ÅÅ·ÏÁÏµç´Å·§
; 模具真空和吹气
741   LD>=    W7 D2112  ; Í¹ÂÖµ±Ç°½Ç¶È / Í¨·çÅÅ³öÆø´ò¿ª½Ç¶È
      AND<=   W7 D2114  ; Í¹ÂÖµ±Ç°½Ç¶È / Í¨·çÅÅ³öÆø¹Ø±Õ½Ç¶È
      LDI     X2E  ; »úÐµÊÖ(ÊÖ¶¯/×Ô¶¯)
      AND     Y11AA  ; ÊÖ¶¯Ä£¾ßÅÅ³öÆøµç´Å·§
      ORB
      AND     L100  ; Ä£¾ßÅÅ³öÆøµç´Å·§ÔÊÐí
      OUT     Y1AA  ; Ä£¾ßÅÅ³öÆøµç´Å·§
752   LD>=    W7 D2120  ; Í¹ÂÖµ±Ç°½Ç¶È / ¸ºÑ¹´ò¿ª½Ç¶È
      AND<=   W7 D2122  ; Í¹ÂÖµ±Ç°½Ç¶È / ¸ºÑ¹¹Ø±Õ½Ç¶È
      LDI     X2E  ; »úÐµÊÖ(ÊÖ¶¯/×Ô¶¯)
      AND     Y11AB  ; ÊÖ¶¯Ä£¾ßÕæ¿Õ·§£¨ÎüÁÏ£©
      ORB
      AND     L101  ; Ä£¾ßÕæ¿Õ·§£¨ÎüÁÏ£©ÔÊÐí
      OUT     Y1AB  ; Ä£¾ßÕæ¿Õ·§£¨ÎüÁÏ£©
763   LD      X2E  ; »úÐµÊÖ(ÊÖ¶¯/×Ô¶¯)
      LD      M199  ; ¿ÕÆ¬²»´µÆø
      OR      M195  ; iu78t
      ANB
      LDI     X2E  ; »úÐµÊÖ(ÊÖ¶¯/×Ô¶¯)
      AND     L4  ; µ÷ÊÔÀëºÏ´µÆø
      ORB
      AND>=   W7 D2116  ; Í¹ÂÖµ±Ç°½Ç¶È / ´µÆø´ò¿ª½Ç¶È
      AND<=   W7 D2118  ; Í¹ÂÖµ±Ç°½Ç¶È / ´µÆø¹Ø±Õ½Ç¶È
      PLS     M105  ; ´µÆø½Ç¶È·¶Î§1PLS
778   LDD=    D18 D2422  ; Öá3µ±Ç°½ø¸øÖµ / ËÍÁÏÖáÊ×³åÇ°Î»ÖÃ
      SET     M195  ; iu78t
782   LDI     X2E  ; »úÐµÊÖ(ÊÖ¶¯/×Ô¶¯)
      RST     M199  ; ¿ÕÆ¬²»´µÆø
      RST     M195  ; iu78t
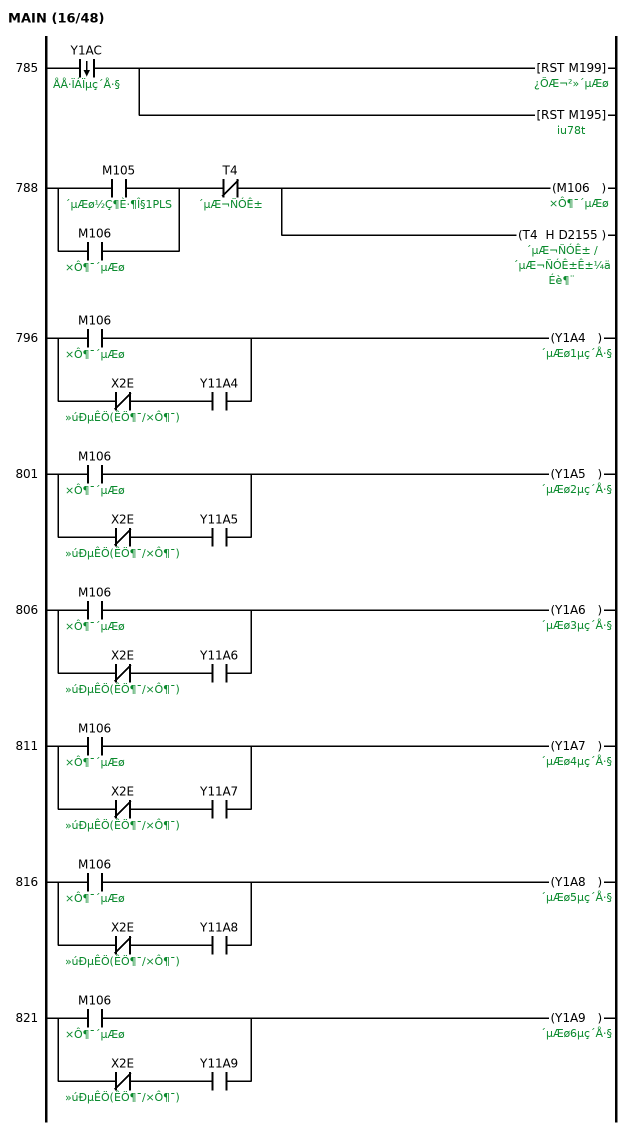
785   LDF     Y1AC  ; ÅÅ·ÏÁÏµç´Å·§
      RST     M199  ; ¿ÕÆ¬²»´µÆø
      RST     M195  ; iu78t
788   LD      M105  ; ´µÆø½Ç¶È·¶Î§1PLS
      OR      M106  ; ×Ô¶¯´µÆø
      ANI     T4  ; ´µÆ¬ÑÓÊ±
      OUT     M106  ; ×Ô¶¯´µÆø
      OUTH    T4 D2155  ; ´µÆ¬ÑÓÊ± / ´µÆ¬ÑÓÊ±Ê±¼äÉè¶¨
796   LD      M106  ; ×Ô¶¯´µÆø
      LDI     X2E  ; »úÐµÊÖ(ÊÖ¶¯/×Ô¶¯)
      AND     Y11A4
      ORB
      OUT     Y1A4  ; ´µÆø1µç´Å·§
801   LD      M106  ; ×Ô¶¯´µÆø
      LDI     X2E  ; »úÐµÊÖ(ÊÖ¶¯/×Ô¶¯)
      AND     Y11A5
      ORB
      OUT     Y1A5  ; ´µÆø2µç´Å·§
806   LD      M106  ; ×Ô¶¯´µÆø
      LDI     X2E  ; »úÐµÊÖ(ÊÖ¶¯/×Ô¶¯)
      AND     Y11A6
      ORB
      OUT     Y1A6  ; ´µÆø3µç´Å·§
811   LD      M106  ; ×Ô¶¯´µÆø
      LDI     X2E  ; »úÐµÊÖ(ÊÖ¶¯/×Ô¶¯)
      AND     Y11A7
      ORB
      OUT     Y1A7  ; ´µÆø4µç´Å·§
816   LD      M106  ; ×Ô¶¯´µÆø
      LDI     X2E  ; »úÐµÊÖ(ÊÖ¶¯/×Ô¶¯)
      AND     Y11A8
      ORB
      OUT     Y1A8  ; ´µÆø5µç´Å·§
821   LD      M106  ; ×Ô¶¯´µÆø
      LDI     X2E  ; »úÐµÊÖ(ÊÖ¶¯/×Ô¶¯)
      AND     Y11A9
      ORB
      OUT     Y1A9  ; ´µÆø6µç´Å·§
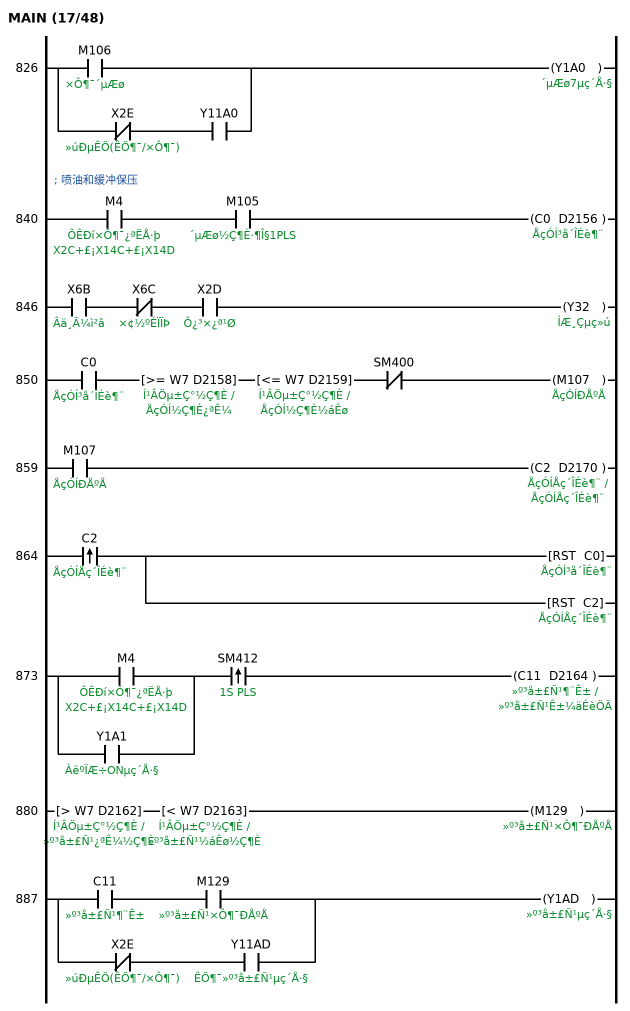
826   LD      M106  ; ×Ô¶¯´µÆø
      LDI     X2E  ; »úÐµÊÖ(ÊÖ¶¯/×Ô¶¯)
      AND     Y11A0
      ORB
      OUT     Y1A0  ; ´µÆø7µç´Å·§
; 喷油和缓冲保压
840   LD      M4  ; ÔÊÐí×Ô¶¯¿ªËÅ·þX2C+£¡X14C+£¡X14D
      AND     M105  ; ´µÆø½Ç¶È·¶Î§1PLS
      OUT     C0 D2156  ; ÅçÓÍ³å´ÎÉè¶¨
846   LD      X6B  ; Âä¸Ã¼ì²â
      ANI     X6C  ; ×¢½ºÉÏÏÞ
      AND     X2D  ; Ô¿³×¿ª¹Ø
      OUT     Y32  ; ÍÆ¸Çµç»ú
850   LD      C0  ; ÅçÓÍ³å´ÎÉè¶¨
      AND>=   W7 D2158  ; Í¹ÂÖµ±Ç°½Ç¶È / ÅçÓÍ½Ç¶È¿ªÊ¼
      AND<=   W7 D2159  ; Í¹ÂÖµ±Ç°½Ç¶È / ÅçÓÍ½Ç¶È½áÊø
      ANI     SM400
      OUT     M107  ; ÅçÓÍÐÅºÅ
859   LD      M107  ; ÅçÓÍÐÅºÅ
      OUT     C2 D2170  ; ÅçÓÍÅç´ÎÉè¶¨ / ÅçÓÍÅç´ÎÉè¶¨
864   LDP     C2  ; ÅçÓÍÅç´ÎÉè¶¨
      RST     C0  ; ÅçÓÍ³å´ÎÉè¶¨
      RST     C2  ; ÅçÓÍÅç´ÎÉè¶¨
873   LD      M4  ; ÔÊÐí×Ô¶¯¿ªËÅ·þX2C+£¡X14C+£¡X14D
      OR      Y1A1  ; ÀëºÏÆ÷ONµç´Å·§
      ANDP    SM412  ; 1S PLS
      OUT     C11 D2164  ; »º³å±£Ñ¹¶¨Ê± / »º³å±£Ñ¹Ê±¼äÉèÖÃ
880   LD>     W7 D2162  ; Í¹ÂÖµ±Ç°½Ç¶È / »º³å±£Ñ¹¿ªÊ¼½Ç¶È
      AND<    W7 D2163  ; Í¹ÂÖµ±Ç°½Ç¶È / »º³å±£Ñ¹½áÊø½Ç¶È
      OUT     M129  ; »º³å±£Ñ¹×Ô¶¯ÐÅºÅ
887   LD      C11  ; »º³å±£Ñ¹¶¨Ê±
      AND     M129  ; »º³å±£Ñ¹×Ô¶¯ÐÅºÅ
      LDI     X2E  ; »úÐµÊÖ(ÊÖ¶¯/×Ô¶¯)
      AND     Y11AD  ; ÊÖ¶¯»º³å±£Ñ¹µç´Å·§
      ORB
      OUT     Y1AD  ; »º³å±£Ñ¹µç´Å·§
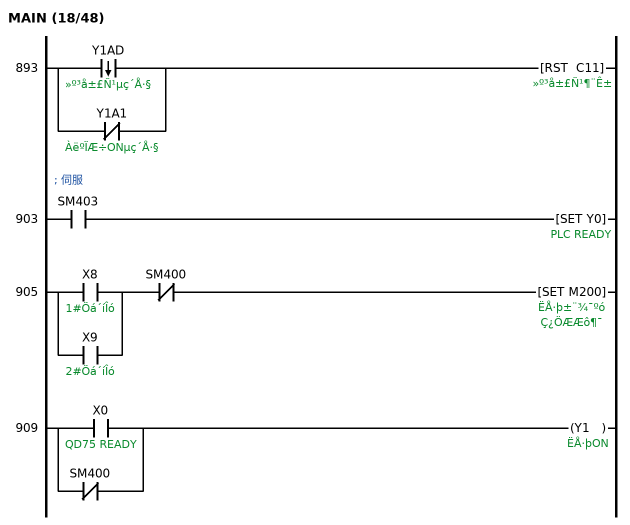
893   LDF     Y1AD  ; »º³å±£Ñ¹µç´Å·§
      ORI     Y1A1  ; ÀëºÏÆ÷ONµç´Å·§
      RST     C11  ; »º³å±£Ñ¹¶¨Ê±
; 伺服
903   LD      SM403
      SET     Y0  ; PLC READY
905   LD      X8  ; 1#Öá´íÎó
      OR      X9  ; 2#Öá´íÎó
      ANI     SM400
      SET     M200  ; ËÅ·þ±¨¾¯ºóÇ¿ÖÆÆô¶¯
909   LD      X0  ; QD75 READY
      ORI     SM400
      OUT     Y1  ; ËÅ·þON
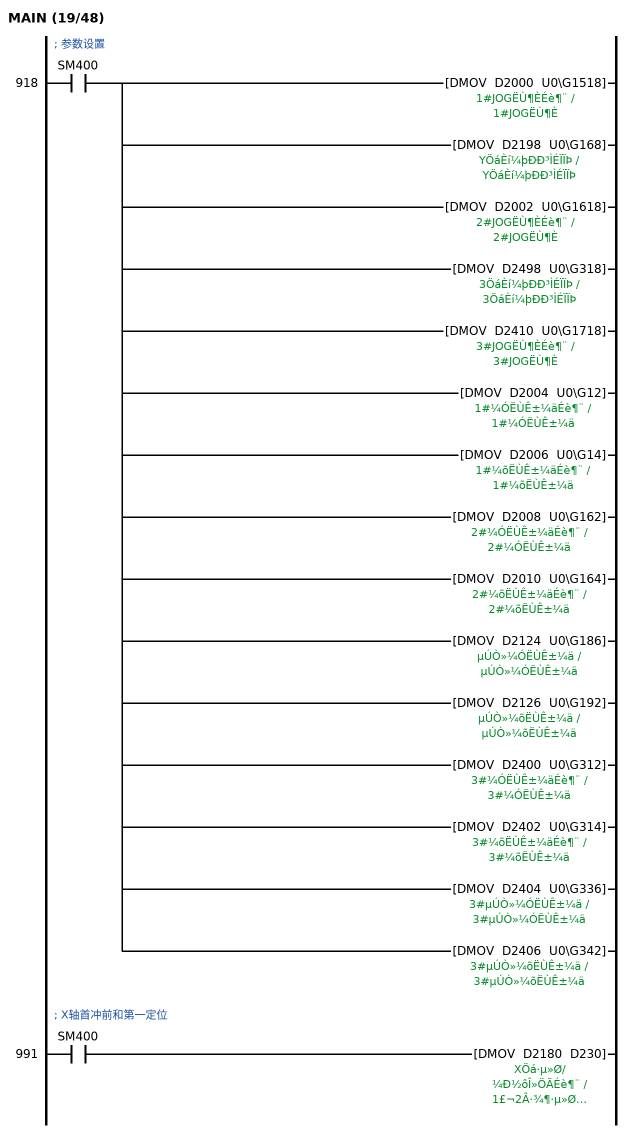
; 参数设置
918   LD      SM400
      DMOV    D2000 U0\G1518  ; 1#JOGËÙ¶ÈÉè¶¨ / 1#JOGËÙ¶È
      DMOV    D2198 U0\G168  ; YÖáÈí¼þÐÐ³ÌÉÏÏÞ / YÖáÈí¼þÐÐ³ÌÉÏÏÞ
      DMOV    D2002 U0\G1618  ; 2#JOGËÙ¶ÈÉè¶¨ / 2#JOGËÙ¶È
      DMOV    D2498 U0\G318  ; 3ÖáÈí¼þÐÐ³ÌÉÏÏÞ / 3ÖáÈí¼þÐÐ³ÌÉÏÏÞ
      DMOV    D2410 U0\G1718  ; 3#JOGËÙ¶ÈÉè¶¨ / 3#JOGËÙ¶È
      DMOV    D2004 U0\G12  ; 1#¼ÓËÙÊ±¼äÉè¶¨ / 1#¼ÓËÙÊ±¼ä
      DMOV    D2006 U0\G14  ; 1#¼õËÙÊ±¼äÉè¶¨ / 1#¼õËÙÊ±¼ä
      DMOV    D2008 U0\G162  ; 2#¼ÓËÙÊ±¼äÉè¶¨ / 2#¼ÓËÙÊ±¼ä
      DMOV    D2010 U0\G164  ; 2#¼õËÙÊ±¼äÉè¶¨ / 2#¼õËÙÊ±¼ä
      DMOV    D2124 U0\G186  ; µÚÒ»¼ÓËÙÊ±¼ä / µÚÒ»¼ÓËÙÊ±¼ä
      DMOV    D2126 U0\G192  ; µÚÒ»¼õËÙÊ±¼ä / µÚÒ»¼õËÙÊ±¼ä
      DMOV    D2400 U0\G312  ; 3#¼ÓËÙÊ±¼äÉè¶¨ / 3#¼ÓËÙÊ±¼ä
      DMOV    D2402 U0\G314  ; 3#¼õËÙÊ±¼äÉè¶¨ / 3#¼õËÙÊ±¼ä
      DMOV    D2404 U0\G336  ; 3#µÚÒ»¼ÓËÙÊ±¼ä / 3#µÚÒ»¼ÓËÙÊ±¼ä
      DMOV    D2406 U0\G342  ; 3#µÚÒ»¼õËÙÊ±¼ä / 3#µÚÒ»¼õËÙÊ±¼ä
; X轴首冲前和第一定位
991   LD      SM400
      DMOV    D2180 D230  ; XÖá·µ»Ø/¼Ð½ôÎ»ÖÃÉè¶¨ / 1£¬2Â·¾¶·µ»Ø/¼Ð½ô¶¨Î»Î»ÖÃ
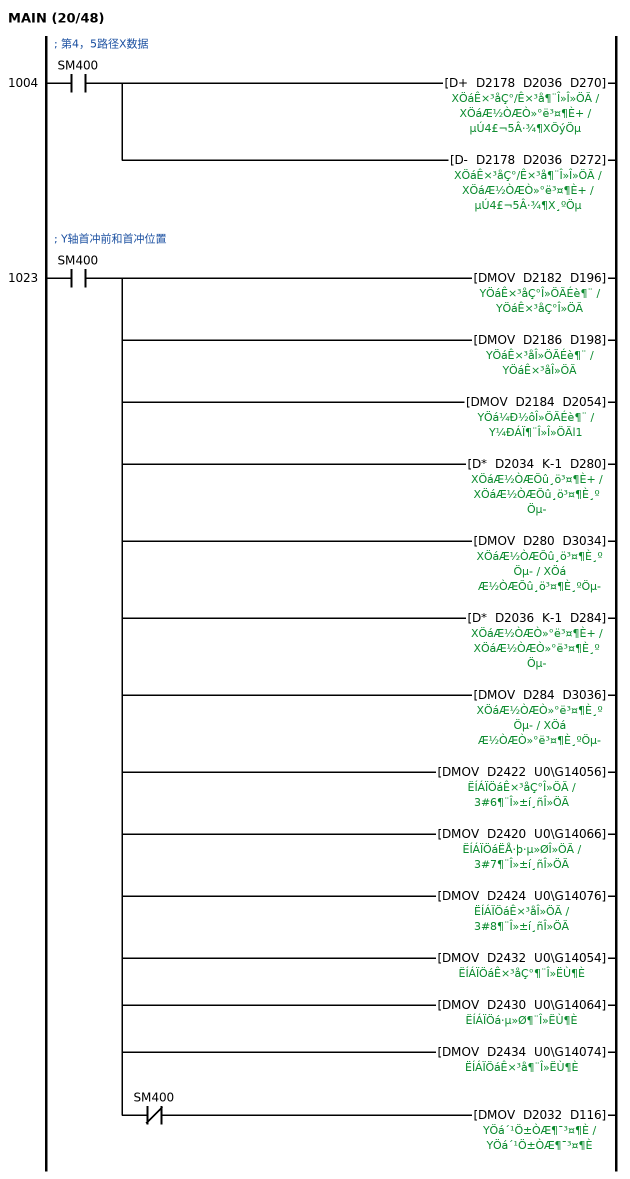
; 第4，5路径X数据
1004  LD      SM400
      D+      D2178 D2036 D270  ; XÖáÊ×³åÇ°/Ê×³å¶¨Î»Î»ÖÃ / XÖáÆ½ÒÆÒ»°ë³¤¶È+ / µÚ4£¬5Â·¾¶XÕýÖµ
      D-      D2178 D2036 D272  ; µÚ4£¬5Â·¾¶X¸ºÖµ
; Y轴首冲前和首冲位置
1023  LD      SM400
      DMOV    D2182 D196  ; YÖáÊ×³åÇ°Î»ÖÃÉè¶¨ / YÖáÊ×³åÇ°Î»ÖÃ
      DMOV    D2186 D198  ; YÖáÊ×³åÎ»ÖÃÉè¶¨ / YÖáÊ×³åÎ»ÖÃ
      DMOV    D2184 D2054  ; YÖá¼Ð½ôÎ»ÖÃÉè¶¨ / Y¼ÐÁÏ¶¨Î»Î»ÖÃl1
      D*      D2034 K-1 D280  ; XÖáÆ½ÒÆÕû¸ö³¤¶È+ / XÖáÆ½ÒÆÕû¸ö³¤¶È¸ºÖµ-
      DMOV    D280 D3034  ; XÖáÆ½ÒÆÕû¸ö³¤¶È¸ºÖµ-
      D*      D2036 K-1 D284  ; XÖáÆ½ÒÆÒ»°ë³¤¶È¸ºÖµ-
      DMOV    D284 D3036  ; XÖáÆ½ÒÆÒ»°ë³¤¶È¸ºÖµ-
      DMOV    D2422 U0\G14056  ; 3#6¶¨Î»±í¸ñÎ»ÖÃ
      DMOV    D2420 U0\G14066  ; ËÍÁÏÖáËÅ·þ·µ»ØÎ»ÖÃ / 3#7¶¨Î»±í¸ñÎ»ÖÃ
      DMOV    D2424 U0\G14076  ; ËÍÁÏÖáÊ×³åÎ»ÖÃ / 3#8¶¨Î»±í¸ñÎ»ÖÃ
      DMOV    D2432 U0\G14054  ; ËÍÁÏÖáÊ×³åÇ°¶¨Î»ËÙ¶È
      DMOV    D2430 U0\G14064  ; ËÍÁÏÖá·µ»Ø¶¨Î»ËÙ¶È
      DMOV    D2434 U0\G14074  ; ËÍÁÏÖáÊ×³å¶¨Î»ËÙ¶È
      ANI     SM400
      DMOV    D2032 D116  ; YÖá´¹Ö±ÒÆ¶¯³¤¶È / YÖá´¹Ö±ÒÆ¶¯³¤¶È
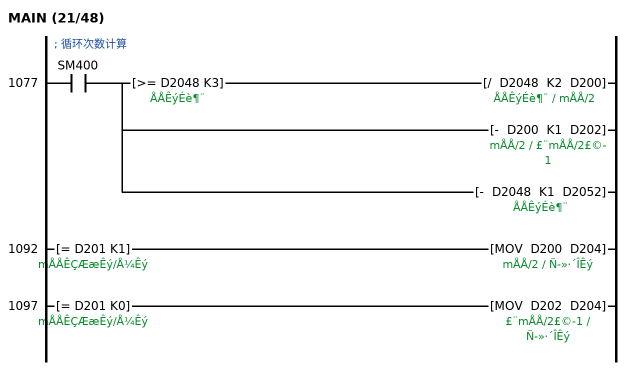
; 循环次数计算
1077  LD      SM400
      MPS
      AND>=   D2048 K3  ; ÅÅÊýÉè¶¨
      /       D2048 K2 D200  ; mÅÅ/2
      MPP
      -       D200 K1 D202  ; £¨mÅÅ/2£©-1
      -       D2048 K1 D2052
1092  LD=     D201 K1  ; mÅÅÊÇÆæÊý/Å¼Êý
      MOV     D200 D204  ; Ñ­»·´ÎÊý
1097  LD=     D201 K0  ; mÅÅÊÇÆæÊý/Å¼Êý
      MOV     D202 D204
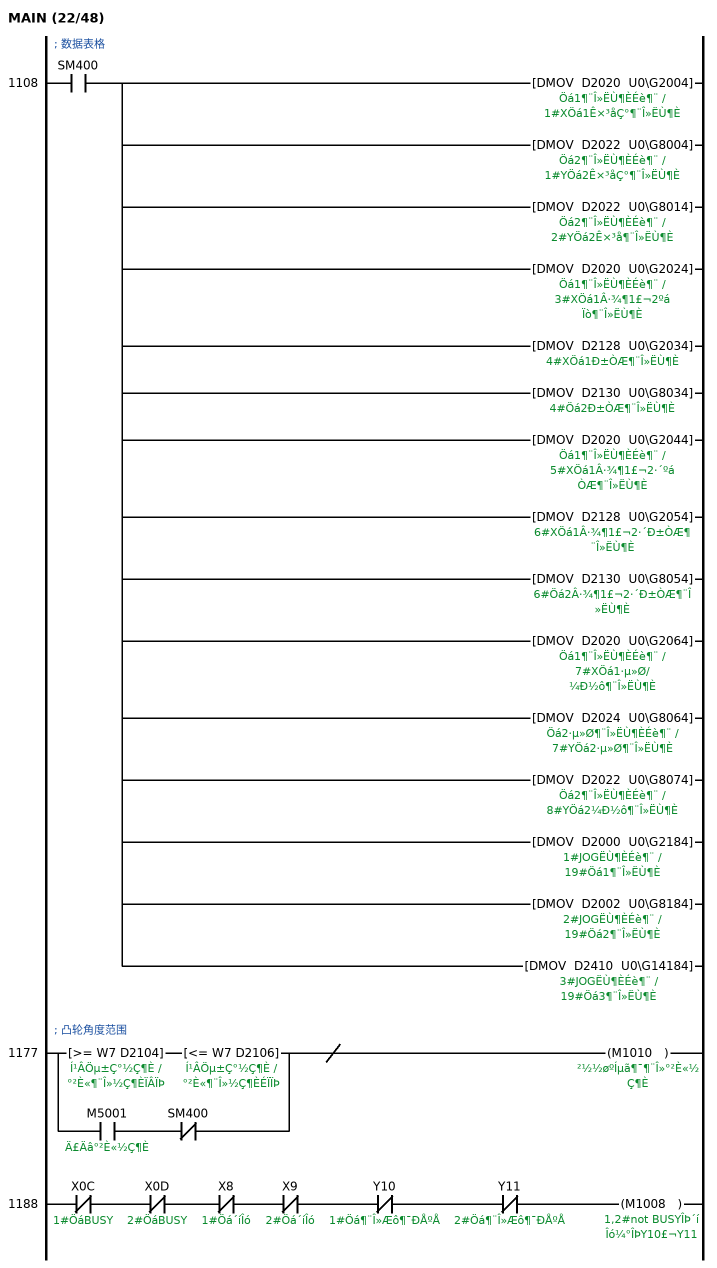
; 数据表格
1108  LD      SM400
      DMOV    D2020 U0\G2004  ; Öá1¶¨Î»ËÙ¶ÈÉè¶¨ / 1#XÖá1Ê×³åÇ°¶¨Î»ËÙ¶È
      DMOV    D2022 U0\G8004  ; Öá2¶¨Î»ËÙ¶ÈÉè¶¨ / 1#YÖá2Ê×³åÇ°¶¨Î»ËÙ¶È
      DMOV    D2022 U0\G8014  ; 2#YÖá2Ê×³å¶¨Î»ËÙ¶È
      DMOV    D2020 U0\G2024  ; 3#XÖá1Â·¾¶1£¬2ºáÏò¶¨Î»ËÙ¶È
      DMOV    D2128 U0\G2034  ; 4#XÖá1Ð±ÒÆ¶¨Î»ËÙ¶È
      DMOV    D2130 U0\G8034  ; 4#Öá2Ð±ÒÆ¶¨Î»ËÙ¶È
      DMOV    D2020 U0\G2044  ; 5#XÖá1Â·¾¶1£¬2·´ºáÒÆ¶¨Î»ËÙ¶È
      DMOV    D2128 U0\G2054  ; 6#XÖá1Â·¾¶1£¬2·´Ð±ÒÆ¶¨Î»ËÙ¶È
      DMOV    D2130 U0\G8054  ; 6#Öá2Â·¾¶1£¬2·´Ð±ÒÆ¶¨Î»ËÙ¶È
      DMOV    D2020 U0\G2064  ; 7#XÖá1·µ»Ø/¼Ð½ô¶¨Î»ËÙ¶È
      DMOV    D2024 U0\G8064  ; Öá2·µ»Ø¶¨Î»ËÙ¶ÈÉè¶¨ / 7#YÖá2·µ»Ø¶¨Î»ËÙ¶È
      DMOV    D2022 U0\G8074  ; 8#YÖá2¼Ð½ô¶¨Î»ËÙ¶È
      DMOV    D2000 U0\G2184  ; 19#Öá1¶¨Î»ËÙ¶È
      DMOV    D2002 U0\G8184  ; 19#Öá2¶¨Î»ËÙ¶È
      DMOV    D2410 U0\G14184  ; 19#Öá3¶¨Î»ËÙ¶È
; 凸轮角度范围
1177  LD>=    W7 D2104  ; Í¹ÂÖµ±Ç°½Ç¶È / °²È«¶¨Î»½Ç¶ÈÏÂÏÞ
      AND<=   W7 D2106  ; Í¹ÂÖµ±Ç°½Ç¶È / °²È«¶¨Î»½Ç¶ÈÉÏÏÞ
      LD      M5001  ; Ä£Äâ°²È«½Ç¶È
      ANI     SM400
      ORB
      INV
      OUT     M1010  ; ²½½øºÍµã¶¯¶¨Î»°²È«½Ç¶È
1188  LDI     X0C  ; 1#ÖáBUSY
      ANI     X0D  ; 2#ÖáBUSY
      ANI     X8  ; 1#Öá´íÎó
      ANI     X9  ; 2#Öá´íÎó
      ANI     Y10  ; 1#Öá¶¨Î»Æô¶¯ÐÅºÅ
      ANI     Y11  ; 2#Öá¶¨Î»Æô¶¯ÐÅºÅ
      OUT     M1008  ; 1,2#not BUSYÎÞ´íÎó¼°ÎÞY10£¬Y11
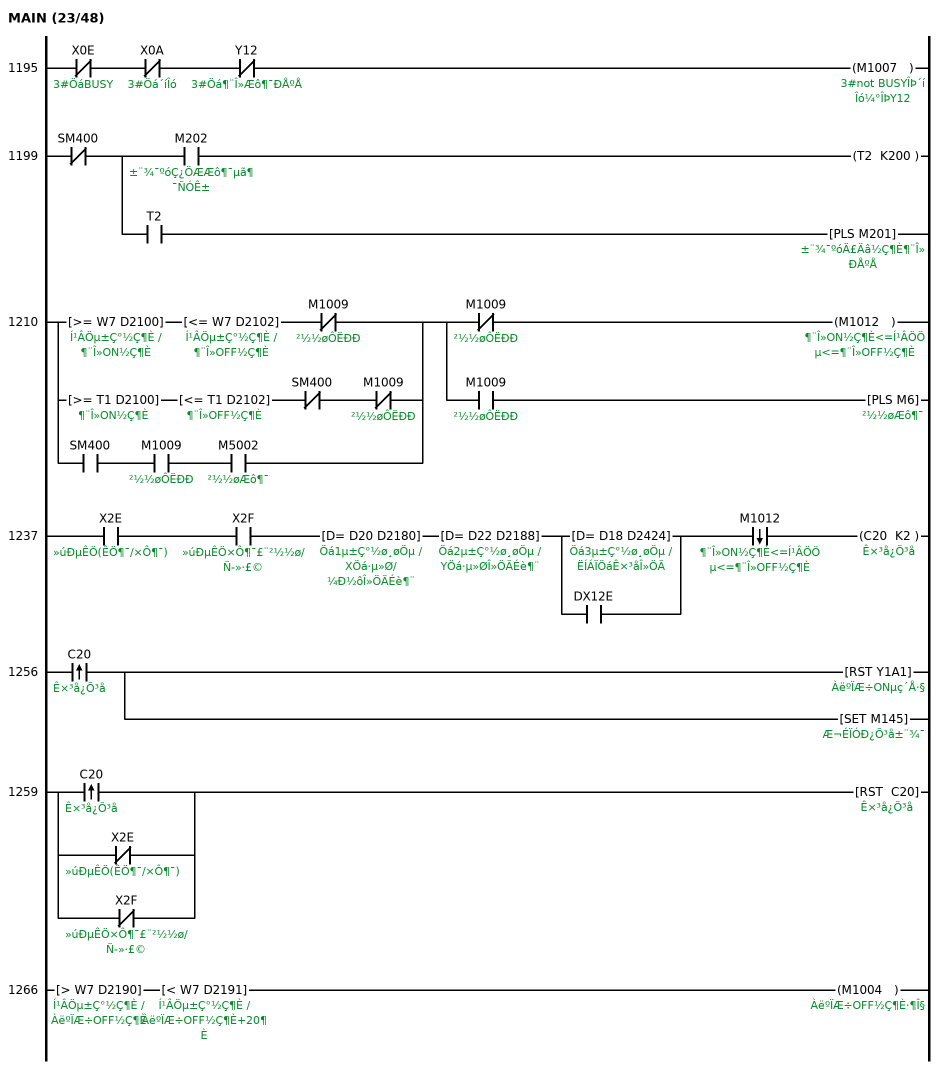
1195  LDI     X0E  ; 3#ÖáBUSY
      ANI     X0A  ; 3#Öá´íÎó
      ANI     Y12  ; 3#Öá¶¨Î»Æô¶¯ÐÅºÅ
      OUT     M1007  ; 3#not BUSYÎÞ´íÎó¼°ÎÞY12
1199  LDI     SM400
      MPS
      AND     M202  ; ±¨¾¯ºóÇ¿ÖÆÆô¶¯µã¶¯ÑÓÊ±
      OUT     T2 K200
      MPP
      AND     T2
      PLS     M201  ; ±¨¾¯ºóÄ£Äâ½Ç¶È¶¨Î»ÐÅºÅ
1210  LD>=    W7 D2100  ; Í¹ÂÖµ±Ç°½Ç¶È / ¶¨Î»ON½Ç¶È
      AND<=   W7 D2102  ; Í¹ÂÖµ±Ç°½Ç¶È / ¶¨Î»OFF½Ç¶È
      ANI     M1009  ; ²½½øÔËÐÐ
      LD>=    T1 D2100  ; ¶¨Î»ON½Ç¶È
      AND<=   T1 D2102  ; ¶¨Î»OFF½Ç¶È
      ANI     SM400
      ANI     M1009  ; ²½½øÔËÐÐ
      ORB
      LD      SM400
      AND     M1009  ; ²½½øÔËÐÐ
      AND     M5002  ; ²½½øÆô¶¯
      ORB
      MPS
      ANI     M1009  ; ²½½øÔËÐÐ
      OUT     M1012  ; ¶¨Î»ON½Ç¶È<=Í¹ÂÖÖµ<=¶¨Î»OFF½Ç¶È
      MPP
      AND     M1009  ; ²½½øÔËÐÐ
      PLS     M6  ; ²½½øÆô¶¯
1237  LD      X2E  ; »úÐµÊÖ(ÊÖ¶¯/×Ô¶¯)
      AND     X2F  ; »úÐµÊÖ×Ô¶¯£¨²½½ø/Ñ­»·£©
      ANDD=   D20 D2180  ; Öá1µ±Ç°½ø¸øÖµ / XÖá·µ»Ø/¼Ð½ôÎ»ÖÃÉè¶¨
      ANDD=   D22 D2188  ; Öá2µ±Ç°½ø¸øÖµ / YÖá·µ»ØÎ»ÖÃÉè¶¨
      LDD=    D18 D2424  ; Öá3µ±Ç°½ø¸øÖµ / ËÍÁÏÖáÊ×³åÎ»ÖÃ
      OR      DX12E
      ANB
      ANDF    M1012  ; ¶¨Î»ON½Ç¶È<=Í¹ÂÖÖµ<=¶¨Î»OFF½Ç¶È
      OUT     C20 K2  ; Ê×³å¿Õ³å
1256  LDP     C20  ; Ê×³å¿Õ³å
      RST     Y1A1  ; ÀëºÏÆ÷ONµç´Å·§
      SET     M145  ; Æ¬ÉÏÓÐ¿Õ³å±¨¾¯
1259  LDP     C20  ; Ê×³å¿Õ³å
      ORI     X2E  ; »úÐµÊÖ(ÊÖ¶¯/×Ô¶¯)
      ORI     X2F  ; »úÐµÊÖ×Ô¶¯£¨²½½ø/Ñ­»·£©
      RST     C20  ; Ê×³å¿Õ³å
1266  LD>     W7 D2190  ; Í¹ÂÖµ±Ç°½Ç¶È / ÀëºÏÆ÷OFF½Ç¶È
      AND<    W7 D2191  ; Í¹ÂÖµ±Ç°½Ç¶È / ÀëºÏÆ÷OFF½Ç¶È+20¶È
      OUT     M1004  ; ÀëºÏÆ÷OFF½Ç¶È·¶Î§
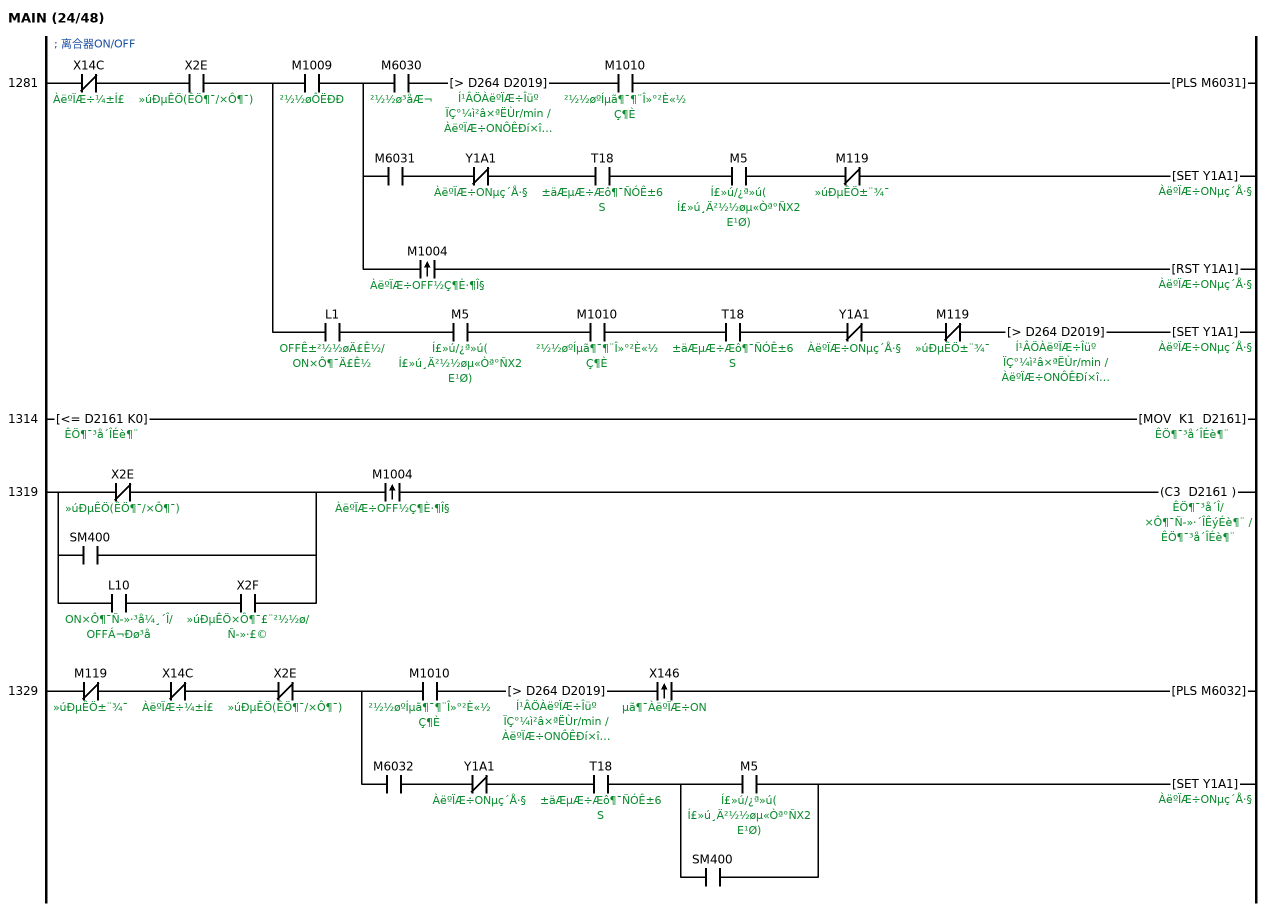
; 离合器ON/OFF
1281  LDI     X14C  ; ÀëºÏÆ÷¼±Í£
      AND     X2E  ; »úÐµÊÖ(ÊÖ¶¯/×Ô¶¯)
      MPS
      AND     M1009  ; ²½½øÔËÐÐ
      MPS
      AND     M6030  ; ²½½ø³åÆ¬
      AND>    D264 D2019  ; Í¹ÂÖÀëºÏÆ÷ÎüºÏÇ°¼ì²â×ªËÙr/min / ÀëºÏÆ÷ONÔÊÐí×îµÍËÙ¶ÈÉè¶¨
      AND     M1010  ; ²½½øºÍµã¶¯¶¨Î»°²È«½Ç¶È
      PLS     M6031
      MRD
      AND     M6031
      ANI     Y1A1  ; ÀëºÏÆ÷ONµç´Å·§
      AND     T18  ; ±äÆµÆ÷Æô¶¯ÑÓÊ±6S
      AND     M5  ; Í£»ú/¿ª»ú(Í£»ú¸Ä²½½øµ«Òª°ÑX2E¹Ø)
      ANI     M119  ; »úÐµÊÖ±¨¾¯
      SET     Y1A1  ; ÀëºÏÆ÷ONµç´Å·§
      MPP
      ANDP    M1004  ; ÀëºÏÆ÷OFF½Ç¶È·¶Î§
      RST     Y1A1  ; ÀëºÏÆ÷ONµç´Å·§
      MPP
      AND     L1  ; OFFÊ±²½½øÄ£Ê½/ON×Ô¶¯Ä£Ê½
      AND     M5  ; Í£»ú/¿ª»ú(Í£»ú¸Ä²½½øµ«Òª°ÑX2E¹Ø)
      AND     M1010  ; ²½½øºÍµã¶¯¶¨Î»°²È«½Ç¶È
      AND     T18  ; ±äÆµÆ÷Æô¶¯ÑÓÊ±6S
      ANI     Y1A1  ; ÀëºÏÆ÷ONµç´Å·§
      ANI     M119  ; »úÐµÊÖ±¨¾¯
      AND>    D264 D2019  ; Í¹ÂÖÀëºÏÆ÷ÎüºÏÇ°¼ì²â×ªËÙr/min / ÀëºÏÆ÷ONÔÊÐí×îµÍËÙ¶ÈÉè¶¨
      SET     Y1A1  ; ÀëºÏÆ÷ONµç´Å·§
1314  LD<=    D2161 K0  ; ÊÖ¶¯³å´ÎÉè¶¨
      MOV     K1 D2161
1319  LDI     X2E  ; »úÐµÊÖ(ÊÖ¶¯/×Ô¶¯)
      OR      SM400
      LD      L10  ; ON×Ô¶¯Ñ­»·³å¼¸´Î/OFFÁ¬Ðø³å
      AND     X2F  ; »úÐµÊÖ×Ô¶¯£¨²½½ø/Ñ­»·£©
      ORB
      ANDP    M1004  ; ÀëºÏÆ÷OFF½Ç¶È·¶Î§
      OUT     C3 D2161  ; ÊÖ¶¯³å´Î/×Ô¶¯Ñ­»·´ÎÊýÉè¶¨ / ÊÖ¶¯³å´ÎÉè¶¨
1329  LDI     M119  ; »úÐµÊÖ±¨¾¯
      ANI     X14C  ; ÀëºÏÆ÷¼±Í£
      ANI     X2E  ; »úÐµÊÖ(ÊÖ¶¯/×Ô¶¯)
      MPS
      AND     M1010  ; ²½½øºÍµã¶¯¶¨Î»°²È«½Ç¶È
      AND>    D264 D2019  ; Í¹ÂÖÀëºÏÆ÷ÎüºÏÇ°¼ì²â×ªËÙr/min / ÀëºÏÆ÷ONÔÊÐí×îµÍËÙ¶ÈÉè¶¨
      ANDP    X146  ; µã¶¯ÀëºÏÆ÷ON
      PLS     M6032
      MPP
      AND     M6032
      ANI     Y1A1  ; ÀëºÏÆ÷ONµç´Å·§
      AND     T18  ; ±äÆµÆ÷Æô¶¯ÑÓÊ±6S
      LD      M5  ; Í£»ú/¿ª»ú(Í£»ú¸Ä²½½øµ«Òª°ÑX2E¹Ø)
      OR      SM400
      ANB
      SET     Y1A1  ; ÀëºÏÆ÷ONµç´Å·§
